C07308=1176.421,-51.106,-43.025,179.479,5.781,149.182
C07309=1176.426,-51.356,-43.013,179.477,5.780,149.183
C07310=1176.431,-51.606,-43.001,179.474,5.780,149.183
C07311=1176.436,-51.856,-42.990,179.472,5.780,149.184
C07312=1176.442,-52.105,-42.979,179.470,5.779,149.185
C07313=1176.447,-52.355,-42.967,179.467,5.779,149.185
C07314=1176.452,-52.605,-42.956,179.465,5.778,149.186
C07315=1176.457,-52.855,-42.944,179.463,5.779,149.187
C07316=1176.462,-53.104,-42.933,179.460,5.778,149.187
C07317=1176.468,-53.354,-42.922,179.458,5.777,149.188
C07318=1176.473,-53.603,-42.910,179.455,5.777,149.188
C07319=1176.477,-53.853,-42.899,179.453,5.777,149.189
C07320=1176.483,-54.103,-42.887,179.451,5.776,149.190
C07321=1176.489,-54.352,-42.877,179.448,5.776,149.190
C07322=1176.494,-54.602,-42.865,179.446,5.776,149.191
C07323=1176.499,-54.852,-42.854,179.444,5.776,149.191
C07324=1176.504,-55.102,-42.842,179.441,5.775,149.192
C07325=1176.509,-55.351,-42.831,179.439,5.774,149.193
C07326=1176.514,-55.600,-42.820,179.437,5.774,149.193
C07327=1176.520,-55.851,-42.808,179.434,5.774,149.194
C07328=1176.524,-56.101,-42.797,179.432,5.774,149.195
C07329=1176.531,-56.350,-42.786,179.430,5.773,149.195
C07330=1176.535,-56.599,-42.774,179.428,5.774,149.196
C07331=1176.540,-56.850,-42.764,179.425,5.773,149.196
C07332=1176.546,-57.099,-42.752,179.423,5.772,149.197
C07333=1176.551,-57.349,-42.741,179.420,5.771,149.198
C07334=1176.556,-57.598,-42.730,179.418,5.772,149.198
C07335=1176.561,-57.849,-42.718,179.416,5.771,149.199
C07336=1176.567,-58.098,-42.708,179.414,5.771,149.199
C07337=1176.572,-58.348,-42.696,179.411,5.770,149.200
C07338=1176.577,-58.597,-42.684,179.409,5.771,149.201
C07339=1176.582,-58.847,-42.674,179.407,5.770,149.201
C07340=1176.588,-59.097,-42.662,179.404,5.769,149.202
C07341=1176.592,-59.346,-42.651,179.402,5.769,149.203
C07342=1176.598,-59.596,-42.641,179.400,5.769,149.203
C07343=1176.603,-59.846,-42.629,179.397,5.769,149.204
C07344=1176.608,-60.095,-42.618,179.395,5.768,149.204
C07345=1176.614,-60.345,-42.607,179.393,5.768,149.205
C07346=1176.618,-60.595,-42.596,179.390,5.768,149.206
C07347=1176.624,-60.845,-42.584,179.388,5.767,149.206
C07348=1176.630,-61.094,-42.574,179.385,5.767,149.207
C07349=1176.634,-61.344,-42.563,179.384,5.766,149.208
C07350=1176.640,-61.594,-42.551,179.381,5.766,149.208
C07351=1176.645,-61.843,-42.541,179.378,5.766,149.209
C07352=1176.650,-62.093,-42.529,179.377,5.766,149.209
C07353=1176.655,-62.343,-42.519,179.374,5.765,149.210
C07354=1176.661,-62.592,-42.507,179.372,5.764,149.211
C07355=1176.666,-62.842,-42.496,179.369,5.764,149.211
C07356=1176.671,-63.092,-42.485,179.367,5.764,149.212
C07357=1176.676,-63.341,-42.474,179.365,5.764,149.212
C07358=1176.682,-63.592,-42.463,179.362,5.763,149.213
C07359=1176.687,-63.841,-42.452,179.360,5.764,149.214
C07360=1176.692,-64.090,-42.441,179.358,5.763,149.214
C07361=1176.697,-64.340,-42.430,179.355,5.762,149.215
C07362=1176.703,-64.590,-42.419,179.354,5.762,149.216
C07363=1176.708,-64.840,-42.408,179.351,5.762,149.216
C07364=1176.712,-65.090,-42.397,179.348,5.762,149.217
C07365=1176.718,-65.339,-42.387,179.346,5.761,149.217
C07366=1176.723,-65.589,-42.376,179.344,5.761,149.218
C07367=1176.729,-65.839,-42.365,179.342,5.760,149.219
C07368=1176.734,-66.088,-42.354,179.339,5.760,149.219
C07369=1176.739,-66.338,-42.343,179.337,5.760,149.220
C07370=1176.744,-66.587,-42.332,179.335,5.759,149.221
C07371=1176.749,-66.838,-42.321,179.332,5.759,149.221
C07372=1176.755,-67.087,-42.310,179.331,5.759,149.222
C07373=1176.760,-67.337,-42.299,179.328,5.759,149.222
C07374=1176.765,-67.586,-42.288,179.325,5.758,149.223
C07375=1176.770,-67.836,-42.278,179.324,5.758,149.224
C07376=1176.776,-68.086,-42.268,179.321,5.758,149.224
C07377=1176.781,-68.335,-42.256,179.319,5.757,149.225
C07378=1176.786,-68.586,-42.245,179.316,5.757,149.225
C07379=1176.792,-68.835,-42.234,179.314,5.757,149.226
C07380=1176.797,-69.085,-42.224,179.312,5.756,149.227
C07381=1176.802,-69.335,-42.213,179.309,5.756,149.227
C07382=1176.807,-69.584,-42.202,179.308,5.756,149.228
C07383=1176.813,-69.834,-42.192,179.305,5.755,149.229
C07384=1176.817,-70.084,-42.181,179.302,5.755,149.229
C07385=1176.823,-70.333,-42.170,179.301,5.755,149.230
C07386=1176.829,-70.584,-42.159,179.298,5.755,149.230
C07387=1176.834,-70.833,-42.148,179.296,5.754,149.231
C07388=1176.839,-71.083,-42.138,179.294,5.754,149.232
C07389=1176.844,-71.332,-42.128,179.291,5.754,149.232
C07390=1176.849,-71.582,-42.116,179.289,5.753,149.233
C07391=1176.855,-71.831,-42.106,179.287,5.753,149.234
C07392=1176.860,-72.082,-42.096,179.285,5.753,149.234
C07393=1176.865,-72.331,-42.085,179.282,5.752,149.235
C07394=1176.870,-72.581,-42.074,179.280,5.753,149.235
C07395=1176.876,-72.830,-42.064,179.278,5.752,149.236
C07396=1176.880,-73.080,-42.053,179.275,5.751,149.237
C07397=1176.886,-73.330,-42.042,179.274,5.751,149.237
C07398=1176.891,-73.580,-42.032,179.271,5.751,149.238
C07399=1176.896,-73.829,-42.021,179.268,5.751,149.239
C07400=1176.902,-74.079,-42.010,179.267,5.751,149.239
C07401=1176.908,-74.329,-41.999,179.264,5.750,149.240
C07402=1176.913,-74.579,-41.989,179.262,5.749,149.240
C07403=1176.918,-74.828,-41.978,179.260,5.750,149.241
C07404=1176.923,-75.078,-41.967,179.257,5.749,149.241
C07405=1176.928,-75.328,-41.957,179.255,5.749,149.242
C07406=1176.934,-75.599,-41.946,179.253,5.749,149.243
C07407=1176.940,-75.869,-41.934,179.250,5.749,149.243
C07408=1176.945,-76.141,-41.923,179.248,5.748,149.244
C07409=1176.951,-76.412,-41.912,179.245,5.747,149.245
C07410=1176.956,-76.661,-41.901,179.243,5.748,149.245
C07411=1176.962,-76.911,-41.891,179.241,5.747,149.246
C07412=1176.967,-77.161,-41.880,179.238,5.747,149.247
C07413=1176.972,-77.411,-41.870,179.236,5.747,149.247
C07414=1176.977,-77.661,-41.859,179.234,5.746,149.248
C07415=1176.983,-77.910,-41.849,179.231,5.746,149.248
C07416=1176.988,-78.160,-41.838,179.230,5.746,149.249
C07417=1176.993,-78.410,-41.828,179.227,5.745,149.250
C07418=1176.999,-78.659,-41.817,179.225,5.745,149.250
C07419=1177.004,-78.909,-41.807,179.223,5.745,149.251
C07420=1177.009,-79.159,-41.797,179.220,5.745,149.252
C07421=1177.014,-79.409,-41.786,179.218,5.744,149.252
C07422=1177.019,-79.658,-41.776,179.216,5.744,149.253
C07423=1177.025,-79.908,-41.766,179.214,5.743,149.253
C07424=1177.030,-80.158,-41.755,179.211,5.743,149.254
C07425=1177.035,-80.407,-41.745,179.209,5.743,149.254
C07426=1177.040,-80.657,-41.734,179.207,5.743,149.255
C07427=1177.046,-80.907,-41.724,179.205,5.743,149.256
C07428=1177.051,-81.156,-41.714,179.202,5.742,149.256
C07429=1177.056,-81.407,-41.703,179.200,5.742,149.257
C07430=1177.062,-81.656,-41.693,179.198,5.742,149.258
C07431=1177.068,-81.906,-41.683,179.196,5.741,149.258
C07432=1177.072,-82.156,-41.673,179.193,5.741,149.259
C07433=1177.077,-82.405,-41.663,179.191,5.741,149.259
C07434=1177.082,-82.655,-41.652,179.189,5.741,149.260
C07435=1177.088,-82.905,-41.642,179.187,5.741,149.261
C07436=1177.094,-83.155,-41.632,179.184,5.740,149.261
C07437=1177.099,-83.405,-41.621,179.182,5.739,149.262
C07438=1177.104,-83.654,-41.611,179.180,5.740,149.263
C07439=1177.109,-83.904,-41.601,179.178,5.739,149.263
C07440=1177.114,-84.154,-41.591,179.175,5.739,149.264
C07441=1177.120,-84.403,-41.580,179.173,5.739,149.264
C07442=1177.125,-84.653,-41.570,179.171,5.738,149.265
C07443=1177.130,-84.903,-41.560,179.169,5.739,149.266
C07444=1177.135,-85.152,-41.550,179.167,5.738,149.266
C07445=1177.141,-85.402,-41.540,179.164,5.737,149.267
C07446=1177.146,-85.652,-41.529,179.162,5.737,149.267
C07447=1177.151,-85.902,-41.519,179.160,5.737,149.268
C07448=1177.157,-86.151,-41.509,179.157,5.736,149.268
C07449=1177.161,-86.401,-41.499,179.155,5.737,149.269
C07450=1177.167,-86.651,-41.489,179.153,5.736,149.270
C07451=1177.172,-86.900,-41.478,179.151,5.736,149.270
C07452=1177.178,-87.150,-41.468,179.148,5.736,149.271
C07453=1177.183,-87.400,-41.459,179.146,5.735,149.272
C07454=1177.188,-87.650,-41.449,179.144,5.735,149.272
C07455=1177.194,-87.899,-41.439,179.142,5.735,149.273
C07456=1177.199,-88.150,-41.428,179.140,5.735,149.273
C07457=1177.204,-88.399,-41.418,179.138,5.734,149.274
C07458=1177.209,-88.648,-41.408,179.135,5.734,149.275
C07459=1177.215,-88.898,-41.398,179.133,5.734,149.275
C07460=1177.220,-89.148,-41.387,179.131,5.733,149.276
C07461=1177.225,-89.398,-41.378,179.129,5.733,149.276
C07462=1177.231,-89.648,-41.368,179.127,5.733,149.277
C07463=1177.236,-89.898,-41.358,179.124,5.733,149.278
C07464=1177.240,-90.147,-41.348,179.122,5.733,149.278
C07465=1177.246,-90.397,-41.338,179.120,5.732,149.279
C07466=1177.252,-90.646,-41.328,179.118,5.732,149.279
C07467=1177.256,-90.897,-41.318,179.115,5.732,149.280
C07468=1177.262,-91.146,-41.308,179.113,5.731,149.281
C07469=1177.267,-91.396,-41.298,179.111,5.732,149.281
C07470=1177.273,-91.645,-41.288,179.109,5.731,149.282
C07471=1177.278,-91.896,-41.278,179.107,5.731,149.283
C07472=1177.283,-92.145,-41.268,179.105,5.730,149.283
C07473=1177.289,-92.395,-41.258,179.102,5.730,149.284
C07474=1177.294,-92.644,-41.248,179.100,5.730,149.284
C07475=1177.300,-92.894,-41.239,179.098,5.730,149.285
C07476=1177.305,-93.145,-41.228,179.096,5.730,149.285
C07477=1177.309,-93.394,-41.219,179.093,5.729,149.286
C07478=1177.315,-93.643,-41.209,179.091,5.729,149.287
C07479=1177.320,-93.893,-41.200,179.089,5.729,149.287
C07480=1177.326,-94.143,-41.189,179.086,5.728,149.288
C07481=1177.331,-94.393,-41.179,179.085,5.728,149.289
C07482=1177.336,-94.642,-41.169,179.082,5.728,149.289
C07483=1177.342,-94.892,-41.160,179.081,5.728,149.290
C07484=1177.347,-95.142,-41.150,179.078,5.728,149.290
C07485=1177.352,-95.391,-41.140,179.076,5.727,149.291
C07486=1177.357,-95.642,-41.130,179.074,5.727,149.292
C07487=1177.362,-95.891,-41.120,179.071,5.726,149.292
C07488=1177.368,-96.141,-41.110,179.069,5.727,149.293
C07489=1177.374,-96.391,-41.101,179.067,5.726,149.293
C07490=1177.379,-96.640,-41.091,179.064,5.726,149.294
C07491=1177.384,-96.890,-41.081,179.063,5.726,149.294
C07492=1177.389,-97.140,-41.072,179.060,5.725,149.295
C07493=1177.394,-97.390,-41.061,179.059,5.725,149.296
C07494=1177.399,-97.640,-41.053,179.056,5.725,149.296
C07495=1177.405,-97.889,-41.042,179.054,5.725,149.297
C07496=1177.411,-98.139,-41.032,179.052,5.725,149.298
C07497=1177.416,-98.389,-41.023,179.049,5.724,149.298
C07498=1177.421,-98.639,-41.013,179.047,5.724,149.299
C07499=1177.426,-98.889,-41.004,179.045,5.723,149.299
C07500=1177.432,-99.138,-40.994,179.043,5.724,149.300
C07501=1177.436,-99.388,-40.984,179.041,5.723,149.300
C07502=1177.442,-99.638,-40.974,179.039,5.723,149.301
C07503=1177.447,-99.887,-40.965,179.037,5.723,149.302
C07504=1177.453,-100.137,-40.955,179.034,5.722,149.302
C07505=1177.458,-100.386,-40.946,179.032,5.722,149.303
C07506=1177.463,-100.637,-40.936,179.030,5.722,149.304
C07507=1177.468,-100.886,-40.926,179.028,5.722,149.304
C07508=1177.474,-101.137,-40.917,179.025,5.722,149.305
C07509=1177.479,-101.386,-40.907,179.024,5.722,149.305
C07510=1177.485,-101.658,-40.896,179.021,5.721,149.306
C07511=1177.491,-101.930,-40.886,179.018,5.721,149.307
C07512=1177.497,-102.201,-40.876,179.016,5.721,149.307
C07513=1177.502,-102.473,-40.865,179.014,5.720,149.308
C07514=1177.508,-102.723,-40.856,179.012,5.720,149.309
C07515=1177.513,-102.972,-40.846,179.010,5.720,149.309
C07516=1177.519,-103.222,-40.837,179.007,5.720,149.310
C07517=1177.523,-103.471,-40.827,179.006,5.720,149.310
C07518=1177.529,-103.722,-40.817,179.003,5.719,149.311
C07519=1177.534,-103.972,-40.808,179.001,5.719,149.311
C07520=1177.539,-104.221,-40.799,178.999,5.719,149.312
C07521=1177.545,-104.471,-40.789,178.996,5.718,149.313
C07522=1177.550,-104.721,-40.780,178.994,5.719,149.313
C07523=1177.555,-104.971,-40.770,178.992,5.718,149.314
C07524=1177.560,-105.220,-40.761,178.990,5.718,149.315
C07525=1177.566,-105.470,-40.751,178.988,5.717,149.315
C07526=1177.571,-105.720,-40.742,178.986,5.718,149.316
C07527=1177.576,-105.969,-40.733,178.984,5.717,149.316
C07528=1177.582,-106.219,-40.723,178.982,5.717,149.317
C07529=1177.587,-106.469,-40.713,178.979,5.717,149.317
C07530=1177.593,-106.719,-40.704,178.978,5.717,149.318
C07531=1177.598,-106.969,-40.695,178.975,5.716,149.319
C07532=1177.603,-107.218,-40.685,178.973,5.716,149.319
C07533=1177.609,-107.468,-40.676,178.971,5.716,149.320
C07534=1177.614,-107.718,-40.667,178.969,5.715,149.320
C07535=1177.619,-107.967,-40.657,178.967,5.716,149.321
C07536=1177.625,-108.217,-40.648,178.964,5.715,149.322
C07537=1177.630,-108.467,-40.639,178.962,5.715,149.322
C07538=1177.635,-108.716,-40.629,178.960,5.714,149.323
C07539=1177.641,-108.967,-40.620,178.958,5.715,149.323
C07540=1177.646,-109.216,-40.611,178.956,5.714,149.324
C07541=1177.651,-109.466,-40.601,178.954,5.714,149.325
C07542=1177.657,-109.716,-40.592,178.952,5.714,149.325
C07543=1177.662,-109.966,-40.583,178.950,5.714,149.326
C07544=1177.667,-110.215,-40.573,178.947,5.713,149.326
C07545=1177.673,-110.465,-40.564,178.946,5.713,149.327
C07546=1177.678,-110.715,-40.555,178.943,5.713,149.328
C07547=1177.683,-110.965,-40.546,178.941,5.712,149.328
C07548=1177.688,-111.214,-40.536,178.939,5.713,149.329
C07549=1177.694,-111.464,-40.527,178.937,5.712,149.329
C07550=1177.699,-111.714,-40.518,178.934,5.712,149.330
C07551=1177.705,-111.964,-40.509,178.932,5.711,149.330
C07552=1177.710,-112.213,-40.499,178.930,5.712,149.331
C07553=1177.715,-112.463,-40.490,178.928,5.711,149.332
C07554=1177.720,-112.713,-40.481,178.926,5.711,149.332
C07555=1177.726,-112.963,-40.472,178.924,5.711,149.333
C07556=1177.731,-113.213,-40.462,178.922,5.711,149.333
C07557=1177.736,-113.462,-40.453,178.919,5.710,149.334
C07558=1177.742,-113.713,-40.444,178.918,5.710,149.335
C07559=1177.747,-113.962,-40.435,178.915,5.710,149.335
C07560=1177.752,-114.212,-40.426,178.914,5.710,149.336
C07561=1177.757,-114.462,-40.417,178.911,5.710,149.336
C07562=1177.763,-114.712,-40.407,178.909,5.710,149.337
C07563=1177.768,-114.961,-40.398,178.907,5.709,149.337
C07564=1177.773,-115.211,-40.389,178.905,5.709,149.338
C07565=1177.778,-115.461,-40.380,178.903,5.709,149.339
C07566=1177.784,-115.710,-40.372,178.901,5.709,149.339
C07567=1177.790,-115.961,-40.362,178.899,5.708,149.340
C07568=1177.795,-116.210,-40.352,178.896,5.709,149.341
C07569=1177.800,-116.460,-40.344,178.894,5.708,149.341
C07570=1177.805,-116.709,-40.335,178.893,5.708,149.342
C07571=1177.810,-116.959,-40.326,178.890,5.707,149.342
C07572=1177.816,-117.209,-40.316,178.888,5.708,149.343
C07573=1177.821,-117.459,-40.307,178.886,5.707,149.343
C07574=1177.827,-117.709,-40.298,178.884,5.707,149.344
C07575=1177.832,-117.959,-40.290,178.881,5.707,149.345
C07576=1177.837,-118.209,-40.281,178.879,5.706,149.345
C07577=1177.843,-118.458,-40.272,178.878,5.706,149.346
C07578=1177.849,-118.708,-40.263,178.875,5.706,149.346
C07579=1177.853,-118.957,-40.253,178.873,5.706,149.347
C07580=1177.859,-119.207,-40.244,178.871,5.705,149.348
C07581=1177.864,-119.457,-40.235,178.869,5.705,149.348
C07582=1177.869,-119.707,-40.226,178.866,5.705,149.349
C07583=1177.874,-119.957,-40.217,178.865,5.705,149.349
C07584=1177.880,-120.207,-40.208,178.863,5.704,149.350
C07585=1177.886,-120.456,-40.199,178.861,5.705,149.350
C07586=1177.891,-120.706,-40.191,178.858,5.704,149.351
C07587=1177.896,-120.956,-40.182,178.856,5.704,149.352
C07588=1177.901,-121.206,-40.173,178.854,5.703,149.352
C07589=1177.906,-121.456,-40.164,178.852,5.704,149.353
C07590=1177.912,-121.705,-40.155,178.850,5.704,149.353
C07591=1177.917,-121.955,-40.146,178.848,5.703,149.354
C07592=1177.923,-122.204,-40.138,178.846,5.704,149.354
C07593=1177.928,-122.455,-40.128,178.844,5.703,149.355
C07594=1177.934,-122.704,-40.119,178.842,5.703,149.355
C07595=1177.939,-122.954,-40.110,178.840,5.702,149.356
C07596=1177.944,-123.204,-40.101,178.838,5.702,149.357
C07597=1177.949,-123.454,-40.092,178.835,5.702,149.357
C07598=1177.955,-123.704,-40.085,178.834,5.702,149.358
C07599=1177.960,-123.954,-40.076,178.832,5.701,149.358
C07600=1177.966,-124.203,-40.067,178.829,5.702,149.359
C07601=1177.971,-124.453,-40.058,178.827,5.701,149.360
C07602=1177.976,-124.703,-40.049,178.825,5.701,149.360
C07603=1177.981,-124.953,-40.040,178.823,5.701,149.361
C07604=1177.987,-125.202,-40.032,178.821,5.701,149.361
C07605=1177.992,-125.452,-40.023,178.819,5.700,149.362
C07606=1177.997,-125.702,-40.014,178.817,5.700,149.362
C07607=1178.002,-125.952,-40.005,178.815,5.700,149.363
C07608=1178.008,-126.201,-39.996,178.813,5.700,149.364
C07609=1178.014,-126.451,-39.988,178.811,5.699,149.364
C07610=1178.019,-126.701,-39.979,178.809,5.700,149.365
C07611=1178.024,-126.951,-39.970,178.806,5.699,149.365
C07612=1178.029,-127.201,-39.961,178.805,5.699,149.366
C07613=1178.035,-127.450,-39.953,178.802,5.699,149.367
C07614=1177.614,-127.462,-39.992,178.799,5.703,149.368
C07615=1177.609,-127.212,-40.001,178.801,5.702,149.368
C07616=1177.604,-126.962,-40.010,178.803,5.703,149.367
C07617=1177.598,-126.712,-40.019,178.805,5.703,149.367
C07618=1177.593,-126.463,-40.028,178.807,5.702,149.366
C07619=1177.587,-126.213,-40.037,178.809,5.703,149.366
C07620=1177.581,-125.962,-40.045,178.811,5.703,149.365
C07621=1177.576,-125.712,-40.054,178.813,5.704,149.364
C07622=1177.570,-125.463,-40.063,178.815,5.704,149.364
C07623=1177.565,-125.213,-40.072,178.818,5.704,149.363
C07624=1177.560,-124.964,-40.081,178.819,5.704,149.363
C07625=1177.555,-124.714,-40.089,178.821,5.705,149.362
C07626=1177.550,-124.464,-40.098,178.823,5.704,149.361
C07627=1177.544,-124.215,-40.107,178.826,5.705,149.361
C07628=1177.539,-123.965,-40.116,178.828,5.705,149.360
C07629=1177.533,-123.715,-40.125,178.830,5.705,149.360
C07630=1177.528,-123.465,-40.134,178.831,5.705,149.359
C07631=1177.523,-123.215,-40.142,178.834,5.706,149.359
C07632=1177.518,-122.965,-40.151,178.836,5.706,149.358
C07633=1177.512,-122.716,-40.159,178.838,5.706,149.357
C07634=1177.507,-122.466,-40.168,178.840,5.706,149.357
C07635=1177.502,-122.216,-40.177,178.842,5.707,149.356
C07636=1177.496,-121.966,-40.186,178.844,5.706,149.356
C07637=1177.491,-121.716,-40.195,178.846,5.707,149.355
C07638=1177.485,-121.466,-40.204,178.848,5.707,149.355
C07639=1177.480,-121.217,-40.213,178.851,5.708,149.354
C07640=1177.474,-120.967,-40.222,178.852,5.707,149.353
C07641=1177.469,-120.717,-40.231,178.855,5.708,149.353
C07642=1177.464,-120.467,-40.240,178.857,5.708,149.352
C07643=1177.459,-120.218,-40.248,178.859,5.708,149.352
C07644=1177.454,-119.968,-40.257,178.861,5.708,149.351
C07645=1177.448,-119.718,-40.267,178.863,5.709,149.351
C07646=1177.443,-119.468,-40.276,178.865,5.709,149.350
C07647=1177.437,-119.219,-40.284,178.867,5.709,149.349
C07648=1177.432,-118.969,-40.293,178.869,5.709,149.349
C07649=1177.427,-118.719,-40.303,178.872,5.710,149.348
C07650=1177.422,-118.470,-40.312,178.873,5.710,149.348
C07651=1177.417,-118.220,-40.321,178.876,5.710,149.347
C07652=1177.411,-117.970,-40.330,178.878,5.710,149.346
C07653=1177.405,-117.720,-40.339,178.880,5.710,149.346
C07654=1177.400,-117.470,-40.348,178.882,5.710,149.345
C07655=1177.395,-117.220,-40.357,178.884,5.711,149.345
C07656=1177.389,-116.971,-40.365,178.886,5.711,149.344
C07657=1177.384,-116.721,-40.374,178.888,5.711,149.344
C07658=1177.378,-116.471,-40.384,178.890,5.711,149.343
C07659=1177.373,-116.221,-40.393,178.893,5.712,149.342
C07660=1177.368,-115.972,-40.402,178.895,5.711,149.342
C07661=1177.363,-115.722,-40.411,178.897,5.712,149.341
C07662=1177.357,-115.472,-40.421,178.898,5.712,149.341
C07663=1177.352,-115.222,-40.429,178.901,5.713,149.340
C07664=1177.347,-114.972,-40.438,178.903,5.713,149.339
C07665=1177.342,-114.722,-40.447,178.905,5.713,149.339
C07666=1177.337,-114.472,-40.456,178.907,5.713,149.338
C07667=1177.331,-114.223,-40.466,178.910,5.713,149.338
C07668=1177.325,-113.974,-40.475,178.911,5.713,149.337
C07669=1177.320,-113.724,-40.484,178.914,5.714,149.336
C07670=1177.315,-113.474,-40.493,178.916,5.714,149.336
C07671=1177.309,-113.224,-40.502,178.918,5.714,149.335
C07672=1177.304,-112.975,-40.512,178.920,5.714,149.335
C07673=1177.299,-112.725,-40.521,178.922,5.715,149.334
C07674=1177.293,-112.475,-40.530,178.925,5.715,149.333
C07675=1177.288,-112.225,-40.539,178.926,5.715,149.333
C07676=1177.283,-111.975,-40.548,178.929,5.715,149.332
C07677=1177.278,-111.726,-40.558,178.931,5.715,149.332
C07678=1177.272,-111.475,-40.567,178.933,5.716,149.331
C07679=1177.267,-111.226,-40.576,178.935,5.716,149.331
C07680=1177.262,-110.976,-40.585,178.937,5.717,149.330
C07681=1177.256,-110.726,-40.595,178.939,5.716,149.329
C07682=1177.251,-110.476,-40.604,178.941,5.717,149.329
C07683=1177.246,-110.227,-40.613,178.943,5.717,149.328
C07684=1177.240,-109.976,-40.622,178.946,5.717,149.328
C07685=1177.235,-109.727,-40.632,178.948,5.717,149.327
C07686=1177.230,-109.477,-40.641,178.950,5.718,149.327
C07687=1177.224,-109.227,-40.650,178.952,5.717,149.326
C07688=1177.219,-108.978,-40.660,178.954,5.718,149.325
C07689=1177.214,-108.728,-40.669,178.956,5.718,149.325
C07690=1177.208,-108.478,-40.678,178.958,5.718,149.324
C07691=1177.203,-108.229,-40.688,178.961,5.719,149.324
C07692=1177.198,-107.979,-40.697,178.963,5.719,149.323
C07693=1177.192,-107.729,-40.706,178.965,5.720,149.322
C07694=1177.187,-107.479,-40.716,178.967,5.719,149.322
C07695=1177.182,-107.230,-40.725,178.969,5.720,149.321
C07696=1177.176,-106.979,-40.734,178.971,5.719,149.321
C07697=1177.171,-106.730,-40.744,178.973,5.720,149.320
C07698=1177.166,-106.480,-40.753,178.976,5.720,149.319
C07699=1177.160,-106.231,-40.763,178.978,5.721,149.319
C07700=1177.155,-105.981,-40.772,178.980,5.720,149.318
C07701=1177.149,-105.731,-40.781,178.982,5.721,149.318
C07702=1177.144,-105.482,-40.791,178.985,5.721,149.317
C07703=1177.139,-105.232,-40.800,178.986,5.721,149.316
C07704=1177.134,-104.982,-40.810,178.989,5.722,149.316
C07705=1177.129,-104.732,-40.819,178.991,5.722,149.315
C07706=1177.123,-104.481,-40.829,178.993,5.723,149.315
C07707=1177.118,-104.232,-40.839,178.995,5.722,149.314
C07708=1177.112,-103.982,-40.848,178.997,5.723,149.314
C07709=1177.108,-103.733,-40.858,178.999,5.722,149.313
C07710=1177.102,-103.483,-40.867,179.001,5.723,149.312
C07711=1177.097,-103.233,-40.877,179.003,5.723,149.312
C07712=1177.092,-102.984,-40.886,179.006,5.724,149.311
C07713=1177.086,-102.734,-40.896,179.008,5.724,149.310
C07714=1177.081,-102.484,-40.905,179.010,5.724,149.310
C07715=1177.075,-102.212,-40.915,179.012,5.724,149.309
C07716=1177.069,-101.940,-40.926,179.015,5.725,149.309
C07717=1177.064,-101.669,-40.937,179.017,5.725,149.308
C07718=1177.058,-101.397,-40.947,179.019,5.725,149.307
C07719=1177.052,-101.147,-40.956,179.022,5.725,149.307
C07720=1177.048,-100.897,-40.966,179.024,5.726,149.306
C07721=1177.042,-100.647,-40.976,179.026,5.726,149.305
C07722=1177.037,-100.398,-40.985,179.028,5.726,149.305
C07723=1177.031,-100.148,-40.995,179.031,5.726,149.304
C07724=1177.026,-99.899,-41.004,179.032,5.726,149.304
C07725=1177.020,-99.648,-41.014,179.035,5.727,149.303
C07726=1177.015,-99.399,-41.023,179.037,5.727,149.303
C07727=1177.010,-99.150,-41.034,179.039,5.727,149.302
C07728=1177.005,-98.899,-41.043,179.041,5.728,149.301
C07729=1177.000,-98.650,-41.053,179.043,5.727,149.301
C07730=1176.995,-98.400,-41.062,179.046,5.728,149.300
C07731=1176.989,-98.150,-41.072,179.048,5.728,149.299
C07732=1176.984,-97.900,-41.081,179.050,5.729,149.299
C07733=1176.978,-97.651,-41.091,179.052,5.728,149.298
C07734=1176.973,-97.401,-41.102,179.054,5.729,149.298
C07735=1176.968,-97.151,-41.111,179.057,5.729,149.297
C07736=1176.962,-96.901,-41.121,179.058,5.729,149.297
C07737=1176.958,-96.652,-41.131,179.061,5.730,149.296
C07738=1176.952,-96.402,-41.140,179.063,5.730,149.295
C07739=1176.947,-96.152,-41.150,179.065,5.730,149.295
C07740=1176.941,-95.903,-41.160,179.067,5.730,149.294
C07741=1176.936,-95.652,-41.170,179.070,5.730,149.293
C07742=1176.931,-95.403,-41.179,179.072,5.731,149.293
C07743=1176.925,-95.153,-41.190,179.074,5.731,149.292
C07744=1176.920,-94.903,-41.199,179.076,5.732,149.292
C07745=1176.915,-94.654,-41.209,179.078,5.731,149.291
C07746=1176.910,-94.404,-41.219,179.080,5.732,149.291
C07747=1176.904,-94.154,-41.228,179.083,5.732,149.290
C07748=1176.899,-93.904,-41.238,179.085,5.732,149.289
C07749=1176.893,-93.655,-41.249,179.087,5.733,149.289
C07750=1176.888,-93.405,-41.258,179.089,5.733,149.288
C07751=1176.883,-93.155,-41.268,179.092,5.733,149.287
C07752=1176.878,-92.905,-41.278,179.093,5.733,149.287
C07753=1176.873,-92.656,-41.288,179.096,5.734,149.286
C07754=1176.867,-92.406,-41.297,179.098,5.734,149.286
C07755=1176.861,-92.156,-41.308,179.100,5.734,149.285
C07756=1176.857,-91.906,-41.318,179.103,5.734,149.284
C07757=1176.851,-91.657,-41.328,179.104,5.734,149.284
C07758=1176.845,-91.406,-41.337,179.107,5.735,149.283
C07759=1176.841,-91.157,-41.347,179.109,5.735,149.283
C07760=1176.836,-90.907,-41.357,179.111,5.735,149.282
C07761=1176.830,-90.657,-41.368,179.114,5.736,149.282
C07762=1176.825,-90.408,-41.377,179.116,5.735,149.281
C07763=1176.819,-90.158,-41.387,179.118,5.736,149.280
C07764=1176.814,-89.908,-41.397,179.121,5.737,149.280
C07765=1176.809,-89.659,-41.407,179.122,5.737,149.279
C07766=1176.804,-89.409,-41.417,179.125,5.737,149.278
C07767=1176.798,-89.160,-41.427,179.126,5.737,149.278
C07768=1176.793,-88.909,-41.438,179.129,5.737,149.277
C07769=1176.788,-88.659,-41.447,179.131,5.738,149.277
C07770=1176.782,-88.410,-41.457,179.133,5.738,149.276
C07771=1176.777,-88.160,-41.468,179.136,5.738,149.275
C07772=1176.773,-87.910,-41.477,179.138,5.738,149.275
C07773=1176.767,-87.661,-41.487,179.140,5.739,149.274
C07774=1176.761,-87.411,-41.498,179.143,5.739,149.274
C07775=1176.756,-87.161,-41.508,179.145,5.739,149.273
C07776=1176.751,-86.912,-41.518,179.147,5.740,149.272
C07777=1176.746,-86.662,-41.528,179.149,5.740,149.272
C07778=1176.741,-86.411,-41.538,179.151,5.740,149.271
C07779=1176.735,-86.162,-41.548,179.154,5.741,149.271
C07780=1176.729,-85.912,-41.558,179.155,5.741,149.270
C07781=1176.725,-85.662,-41.568,179.158,5.741,149.269
C07782=1176.719,-85.413,-41.579,179.161,5.741,149.269
C07783=1176.714,-85.163,-41.589,179.162,5.741,149.268
C07784=1176.708,-84.914,-41.599,179.165,5.742,149.267
C07785=1176.703,-84.664,-41.610,179.167,5.742,149.267
C07786=1176.698,-84.414,-41.619,179.169,5.742,149.266
C07787=1176.693,-84.165,-41.629,179.171,5.743,149.266
C07788=1176.688,-83.915,-41.640,179.173,5.743,149.265
C07789=1176.682,-83.665,-41.650,179.176,5.743,149.265
C07790=1176.677,-83.415,-41.661,179.178,5.744,149.264
C07791=1176.672,-83.165,-41.670,179.180,5.743,149.263
C07792=1176.667,-82.916,-41.681,179.183,5.744,149.263
C07793=1176.662,-82.666,-41.691,179.185,5.744,149.262
C07794=1176.656,-82.416,-41.701,179.187,5.744,149.262
C07795=1176.651,-82.167,-41.712,179.190,5.745,149.261
C07796=1176.646,-81.916,-41.722,179.191,5.745,149.260
C07797=1176.640,-81.667,-41.732,179.194,5.745,149.260
C07798=1176.635,-81.418,-41.742,179.196,5.746,149.259
C07799=1176.630,-81.167,-41.753,179.198,5.746,149.258
C07800=1176.625,-80.918,-41.763,179.201,5.746,149.258
C07801=1176.620,-80.668,-41.773,179.203,5.747,149.257
C07802=1176.614,-80.418,-41.784,179.205,5.746,149.257
C07803=1176.609,-80.169,-41.794,179.207,5.747,149.256
C07804=1176.604,-79.919,-41.805,179.209,5.747,149.255
C07805=1176.598,-79.669,-41.815,179.211,5.748,149.255
C07806=1176.592,-79.420,-41.825,179.214,5.748,149.254
C07807=1176.587,-79.170,-41.836,179.216,5.748,149.253
C07808=1176.583,-78.920,-41.846,179.218,5.748,149.253
C07809=1176.578,-78.670,-41.856,179.221,5.749,149.252
C07810=1176.572,-78.421,-41.866,179.223,5.749,149.252
C07811=1176.566,-78.171,-41.877,179.225,5.749,149.251
C07812=1176.562,-77.921,-41.888,179.228,5.750,149.251
C07813=1176.556,-77.672,-41.898,179.230,5.750,149.250
C07814=1176.551,-77.422,-41.909,179.232,5.750,149.249
C07815=1176.546,-77.172,-41.919,179.234,5.751,149.249
C07816=1176.541,-76.922,-41.929,179.237,5.750,149.248
C07817=1176.535,-76.672,-41.940,179.239,5.751,149.247
C07818=1176.530,-76.423,-41.951,179.241,5.752,149.247
C07819=1176.524,-76.152,-41.962,179.243,5.751,149.246
C07820=1176.519,-75.880,-41.973,179.246,5.752,149.246
C07821=1176.512,-75.610,-41.985,179.248,5.752,149.245
C07822=1176.507,-75.339,-41.996,179.251,5.753,149.244
C07823=1176.501,-75.088,-42.007,179.253,5.752,149.243
C07824=1176.496,-74.839,-42.017,179.255,5.753,149.243
C07825=1176.490,-74.590,-42.028,179.258,5.754,149.242
C07826=1176.485,-74.340,-42.039,179.260,5.754,149.242
C07827=1176.480,-74.090,-42.049,179.262,5.754,149.241
C07828=1176.475,-73.840,-42.060,179.265,5.754,149.240
C07829=1176.470,-73.591,-42.070,179.266,5.754,149.240
C07830=1176.465,-73.341,-42.081,179.269,5.755,149.239
C07831=1176.459,-73.091,-42.091,179.271,5.756,149.239
C07832=1176.454,-72.841,-42.103,179.273,5.755,149.238
C07833=1176.449,-72.592,-42.113,179.276,5.756,149.238
C07834=1176.444,-72.342,-42.123,179.278,5.756,149.237
C07835=1176.438,-72.092,-42.134,179.280,5.756,149.236
C07836=1176.433,-71.842,-42.145,179.283,5.757,149.236
C07837=1176.428,-71.593,-42.155,179.285,5.757,149.235
C07838=1176.423,-71.343,-42.166,179.287,5.757,149.234
C07839=1176.418,-71.094,-42.177,179.289,5.758,149.234
C07840=1176.413,-70.844,-42.187,179.292,5.758,149.233
C07841=1176.406,-70.594,-42.198,179.294,5.758,149.233
C07842=1176.402,-70.344,-42.209,179.296,5.759,149.232
C07843=1176.396,-70.094,-42.219,179.299,5.759,149.231
C07844=1176.391,-69.845,-42.231,179.301,5.759,149.231
C07845=1176.386,-69.595,-42.241,179.303,5.759,149.230
C07846=1176.381,-69.345,-42.251,179.306,5.760,149.229
C07847=1176.375,-69.096,-42.262,179.308,5.760,149.229
C07848=1176.370,-68.846,-42.273,179.310,5.761,149.228
C07849=1176.364,-68.597,-42.285,179.312,5.761,149.228
C07850=1176.359,-68.346,-42.295,179.315,5.761,149.227
C07851=1176.354,-68.096,-42.306,179.317,5.761,149.226
C07852=1176.349,-67.847,-42.317,179.319,5.762,149.226
C07853=1176.344,-67.597,-42.327,179.322,5.763,149.225
C07854=1176.339,-67.348,-42.338,179.324,5.762,149.224
C07855=1176.334,-67.098,-42.349,179.326,5.763,149.224
C07856=1176.328,-66.849,-42.360,179.329,5.763,149.223
C07857=1176.323,-66.598,-42.371,179.331,5.763,149.223
C07858=1176.317,-66.349,-42.382,179.333,5.764,149.222
C07859=1176.312,-66.099,-42.392,179.335,5.764,149.221
C07860=1176.308,-65.850,-42.404,179.338,5.764,149.221
C07861=1176.301,-65.600,-42.414,179.340,5.765,149.220
C07862=1176.297,-65.350,-42.426,179.342,5.765,149.220
C07863=1176.291,-65.101,-42.436,179.345,5.766,149.219
C07864=1176.286,-64.851,-42.447,179.347,5.765,149.218
C07865=1176.281,-64.601,-42.458,179.349,5.766,149.218
C07866=1176.275,-64.351,-42.469,179.352,5.767,149.217
C07867=1176.270,-64.101,-42.480,179.354,5.766,149.216
C07868=1176.265,-63.852,-42.491,179.356,5.767,149.216
C07869=1176.260,-63.602,-42.501,179.358,5.768,149.215
C07870=1176.255,-63.352,-42.513,179.361,5.767,149.215
C07871=1176.249,-63.103,-42.523,179.363,5.768,149.214
C07872=1176.244,-62.853,-42.535,179.365,5.768,149.213
C07873=1176.240,-62.603,-42.546,179.368,5.769,149.213
C07874=1176.233,-62.353,-42.557,179.370,5.769,149.212
C07875=1176.229,-62.104,-42.568,179.372,5.769,149.211
C07876=1176.223,-61.854,-42.578,179.375,5.770,149.211
C07877=1176.218,-61.605,-42.590,179.377,5.770,149.210
C07878=1176.213,-61.355,-42.601,179.379,5.770,149.210
C07879=1176.207,-61.105,-42.612,179.381,5.771,149.209
C07880=1176.203,-60.856,-42.623,179.384,5.771,149.208
C07881=1176.197,-60.606,-42.635,179.386,5.771,149.208
C07882=1176.192,-60.356,-42.645,179.388,5.772,149.207
C07883=1176.187,-60.106,-42.656,179.391,5.772,149.207
C07884=1176.182,-59.857,-42.668,179.393,5.772,149.206
C07885=1176.176,-59.607,-42.678,179.395,5.773,149.205
C07886=1176.171,-59.357,-42.690,179.397,5.773,149.205
C07887=1176.167,-59.108,-42.701,179.400,5.774,149.204
C07888=1176.160,-58.858,-42.712,179.402,5.773,149.203
C07889=1176.155,-58.608,-42.723,179.404,5.774,149.203
C07890=1176.151,-58.359,-42.734,179.407,5.775,149.202
C07891=1176.145,-58.108,-42.746,179.410,5.775,149.202
C07892=1176.140,-57.859,-42.756,179.411,5.775,149.201
C07893=1176.135,-57.609,-42.768,179.414,5.775,149.200
C07894=1176.130,-57.360,-42.780,179.416,5.776,149.200
C07895=1176.124,-57.110,-42.790,179.418,5.776,149.199
C07896=1176.119,-56.860,-42.802,179.421,5.776,149.198
C07897=1176.114,-56.610,-42.813,179.423,5.777,149.198
C07898=1176.109,-56.361,-42.824,179.426,5.777,149.197
C07899=1176.103,-56.111,-42.835,179.428,5.777,149.197
C07900=1176.098,-55.861,-42.846,179.430,5.778,149.196
C07901=1176.094,-55.612,-42.858,179.433,5.778,149.195
C07902=1176.087,-55.362,-42.869,179.435,5.779,149.195
C07903=1176.083,-55.113,-42.881,179.437,5.779,149.194
C07904=1176.077,-54.862,-42.892,179.440,5.779,149.194
C07905=1176.072,-54.613,-42.903,179.442,5.780,149.193
C07906=1176.066,-54.363,-42.915,179.445,5.780,149.192
C07907=1176.062,-54.114,-42.926,179.447,5.780,149.192
C07908=1176.057,-53.864,-42.937,179.449,5.781,149.191
C07909=1176.052,-53.614,-42.949,179.451,5.781,149.190
C07910=1176.046,-53.365,-42.959,179.454,5.782,149.190
C07911=1176.040,-53.115,-42.971,179.456,5.782,149.189
C07912=1176.036,-52.865,-42.982,179.458,5.782,149.189
C07913=1176.030,-52.615,-42.994,179.461,5.783,149.188
C07914=1176.026,-52.366,-43.006,179.463,5.783,149.187
C07915=1176.020,-52.116,-43.017,179.465,5.783,149.187
C07916=1176.015,-51.867,-43.028,179.467,5.784,149.186
C07917=1176.010,-51.617,-43.040,179.470,5.784,149.186
C07918=1176.005,-51.367,-43.052,179.472,5.785,149.185
C07919=1175.999,-51.118,-43.063,179.474,5.785,149.184
C07920=1175.994,-50.868,-43.074,179.477,5.785,149.184
C07921=1175.988,-50.618,-43.085,179.479,5.786,149.183
C07922=1175.984,-50.368,-43.097,179.482,5.786,149.182
C07923=1175.978,-50.098,-43.109,179.485,5.787,149.182
C07924=1175.972,-49.827,-43.122,179.487,5.787,149.181
C07925=1175.967,-49.557,-43.135,179.489,5.787,149.180
C07926=1175.961,-49.287,-43.146,179.491,5.788,149.180
C07927=1175.956,-49.037,-43.158,179.494,5.788,149.179
C07928=1175.951,-48.787,-43.170,179.497,5.788,149.178
C07929=1175.945,-48.537,-43.182,179.499,5.789,149.178
C07930=1175.940,-48.288,-43.193,179.501,5.789,149.177
C07931=1175.934,-48.039,-43.204,179.504,5.789,149.177
C07932=1175.930,-47.789,-43.216,179.506,5.790,149.176
C07933=1175.924,-47.539,-43.228,179.509,5.790,149.175
C07934=1175.920,-47.290,-43.240,179.511,5.791,149.175
C07935=1175.914,-47.040,-43.251,179.513,5.791,149.174
C07936=1175.909,-46.790,-43.263,179.516,5.791,149.174
C07937=1175.904,-46.540,-43.275,179.518,5.792,149.173
C07938=1175.898,-46.291,-43.286,179.520,5.793,149.172
C07939=1175.894,-46.042,-43.297,179.522,5.792,149.172
C07940=1175.888,-45.792,-43.309,179.525,5.793,149.171
C07941=1175.883,-45.542,-43.321,179.527,5.793,149.170
C07942=1175.878,-45.292,-43.332,179.530,5.794,149.170
C07943=1175.873,-45.042,-43.344,179.532,5.795,149.169
C07944=1175.867,-44.792,-43.356,179.534,5.794,149.169
C07945=1175.862,-44.543,-43.368,179.537,5.795,149.168
C07946=1175.857,-44.294,-43.380,179.539,5.796,149.167
C07947=1175.852,-44.044,-43.391,179.542,5.796,149.167
C07948=1175.847,-43.794,-43.403,179.544,5.796,149.166
C07949=1175.841,-43.544,-43.415,179.546,5.796,149.166
C07950=1175.837,-43.295,-43.426,179.549,5.797,149.165
C07951=1175.831,-43.045,-43.438,179.551,5.798,149.164
C07952=1175.826,-42.795,-43.450,179.554,5.798,149.164
C07953=1175.821,-42.546,-43.462,179.556,5.799,149.163
C07954=1175.816,-42.296,-43.474,179.558,5.799,149.162
C07955=1175.810,-42.046,-43.486,179.560,5.799,149.162
C07956=1175.805,-41.796,-43.498,179.563,5.799,149.161
C07957=1175.800,-41.547,-43.508,179.565,5.800,149.161
C07958=1175.795,-41.298,-43.521,179.568,5.801,149.160
C07959=1175.789,-41.048,-43.533,179.570,5.800,149.159
C07960=1175.784,-40.798,-43.544,179.572,5.801,149.159
C07961=1175.779,-40.548,-43.556,179.575,5.802,149.158
C07962=1175.774,-40.299,-43.569,179.578,5.802,149.157
C07963=1175.768,-40.049,-43.581,179.580,5.803,149.157
C07964=1175.764,-39.800,-43.592,179.582,5.802,149.156
C07965=1175.758,-39.550,-43.604,179.584,5.803,149.156
C07966=1175.753,-39.300,-43.616,179.587,5.804,149.155
C07967=1175.748,-39.050,-43.628,179.589,5.804,149.154
C07968=1175.743,-38.801,-43.640,179.591,5.805,149.154
C07969=1175.738,-38.551,-43.652,179.594,5.805,149.153
C07970=1175.733,-38.301,-43.664,179.596,5.805,149.152
C07971=1175.727,-38.052,-43.676,179.598,5.806,149.152
C07972=1175.722,-37.802,-43.688,179.601,5.806,149.151
C07973=1175.717,-37.553,-43.700,179.604,5.807,149.151
C07974=1175.712,-37.303,-43.712,179.606,5.807,149.150
C07975=1175.706,-37.053,-43.724,179.608,5.807,149.149
C07976=1175.701,-36.803,-43.736,179.611,5.808,149.149
C07977=1175.696,-36.553,-43.748,179.613,5.808,149.148
C07978=1175.691,-36.304,-43.760,179.615,5.809,149.147
C07979=1175.686,-36.055,-43.772,179.618,5.809,149.147
C07980=1175.681,-35.805,-43.784,179.620,5.810,149.146
C07981=1175.676,-35.555,-43.796,179.622,5.810,149.146
C07982=1175.670,-35.305,-43.808,179.625,5.810,149.145
C07983=1175.665,-35.056,-43.821,179.627,5.811,149.144
C07984=1175.660,-34.806,-43.833,179.630,5.811,149.144
C07985=1175.655,-34.556,-43.844,179.632,5.812,149.143
C07986=1175.650,-34.307,-43.857,179.635,5.813,149.143
C07987=1175.644,-34.057,-43.869,179.637,5.812,149.142
C07988=1175.639,-33.808,-43.881,179.639,5.813,149.141
C07989=1175.634,-33.558,-43.893,179.642,5.813,149.141
C07990=1175.629,-33.309,-43.906,179.644,5.814,149.140
C07991=1175.623,-33.059,-43.918,179.646,5.815,149.140
C07992=1175.618,-32.809,-43.930,179.649,5.815,149.139
C07993=1175.613,-32.560,-43.941,179.651,5.815,149.138
C07994=1175.608,-32.310,-43.953,179.653,5.816,149.138
C07995=1175.603,-32.060,-43.966,179.656,5.816,149.137
C07996=1175.597,-31.811,-43.978,179.659,5.817,149.136
C07997=1175.592,-31.561,-43.990,179.661,5.817,149.136
C07998=1175.588,-31.311,-44.003,179.664,5.818,149.135
C07999=1175.582,-31.061,-44.015,179.666,5.818,149.134
C08000=1175.577,-30.812,-44.028,179.668,5.818,149.134
C08001=1175.572,-30.562,-44.040,179.670,5.819,149.133
C08002=1175.567,-30.313,-44.052,179.673,5.819,149.133
C08003=1175.561,-30.063,-44.064,179.675,5.820,149.132
C08004=1175.556,-29.813,-44.077,179.678,5.820,149.131
C08005=1175.551,-29.564,-44.089,179.681,5.821,149.131
C08006=1175.546,-29.314,-44.101,179.683,5.822,149.130
C08007=1175.540,-29.065,-44.114,179.685,5.821,149.130
C08008=1175.536,-28.814,-44.126,179.688,5.822,149.129
C08009=1175.530,-28.565,-44.139,179.690,5.823,149.128
C08010=1175.525,-28.315,-44.151,179.692,5.823,149.128
C08011=1175.520,-28.066,-44.163,179.695,5.823,149.127
C08012=1175.515,-27.816,-44.176,179.697,5.824,149.126
C08013=1175.509,-27.566,-44.188,179.700,5.825,149.126
C08014=1175.504,-27.317,-44.200,179.702,5.826,149.125
C08015=1175.499,-27.068,-44.213,179.704,5.825,149.125
C08016=1175.494,-26.817,-44.225,179.707,5.826,149.124
C08017=1175.489,-26.568,-44.238,179.709,5.826,149.123
C08018=1175.484,-26.318,-44.250,179.712,5.827,149.123
C08019=1175.479,-26.069,-44.262,179.714,5.827,149.122
C08020=1175.473,-25.819,-44.275,179.716,5.828,149.122
C08021=1175.468,-25.570,-44.288,179.719,5.829,149.121
C08022=1175.464,-25.319,-44.300,179.722,5.829,149.120
C08023=1175.458,-25.070,-44.312,179.723,5.829,149.120
C08024=1175.453,-24.821,-44.325,179.726,5.829,149.119
C08025=1175.448,-24.571,-44.338,179.729,5.830,149.118
C08026=1175.443,-24.321,-44.349,179.731,5.831,149.118
C08027=1175.437,-24.051,-44.364,179.734,5.831,149.117
C08028=1175.432,-23.782,-44.377,179.736,5.832,149.116
C08029=1175.426,-23.513,-44.391,179.739,5.832,149.116
C08030=1175.420,-23.242,-44.404,179.742,5.833,149.115
C08031=1175.415,-22.993,-44.417,179.744,5.833,149.114
C08032=1175.410,-22.743,-44.429,179.746,5.834,149.114
C08033=1175.406,-22.493,-44.442,179.749,5.834,149.113
C08034=1175.400,-22.243,-44.454,179.751,5.835,149.113
C08035=1175.395,-21.994,-44.467,179.754,5.835,149.112
C08036=1175.390,-21.745,-44.480,179.757,5.836,149.111
C08037=1175.384,-21.495,-44.493,179.759,5.837,149.111
C08038=1175.379,-21.245,-44.506,179.761,5.836,149.110
C08039=1175.374,-20.996,-44.518,179.763,5.837,149.109
C08040=1175.369,-20.746,-44.530,179.766,5.838,149.109
C08041=1175.364,-20.496,-44.543,179.768,5.838,149.108
C08042=1175.359,-20.246,-44.556,179.771,5.839,149.108
C08043=1175.353,-19.997,-44.569,179.773,5.839,149.107
C08044=1175.348,-19.748,-44.582,179.776,5.840,149.106
C08045=1175.343,-19.498,-44.594,179.778,5.840,149.106
C08046=1175.339,-19.248,-44.607,179.781,5.841,149.105
C08047=1175.334,-18.999,-44.620,179.783,5.842,149.105
C08048=1175.328,-18.749,-44.633,179.786,5.842,149.104
C08049=1175.322,-18.499,-44.645,179.788,5.842,149.103
C08050=1175.318,-18.249,-44.658,179.790,5.842,149.103
C08051=1175.313,-18.000,-44.670,179.793,5.843,149.102
C08052=1175.307,-17.750,-44.684,179.795,5.844,149.102
C08053=1175.302,-17.501,-44.696,179.798,5.844,149.101
C08054=1175.297,-17.251,-44.709,179.800,5.845,149.100
C08055=1175.292,-17.002,-44.722,179.803,5.846,149.100
C08056=1175.286,-16.752,-44.735,179.805,5.846,149.099
C08057=1175.282,-16.502,-44.748,179.808,5.846,149.098
C08058=1175.276,-16.253,-44.760,179.810,5.847,149.098
C08059=1175.271,-16.003,-44.773,179.813,5.848,149.097
C08060=1175.266,-15.753,-44.787,179.815,5.848,149.096
C08061=1175.261,-15.504,-44.799,179.818,5.849,149.096
C08062=1175.256,-15.254,-44.812,179.820,5.849,149.095
C08063=1175.251,-15.004,-44.825,179.822,5.849,149.095
C08064=1175.245,-14.755,-44.838,179.824,5.850,149.094
C08065=1175.240,-14.505,-44.851,179.827,5.850,149.093
C08066=1175.236,-14.255,-44.864,179.830,5.851,149.093
C08067=1175.230,-14.006,-44.877,179.832,5.852,149.092
C08068=1175.225,-13.757,-44.890,179.835,5.852,149.092
C08069=1175.221,-13.507,-44.903,179.837,5.853,149.091
C08070=1175.215,-13.257,-44.916,179.839,5.853,149.090
C08071=1175.210,-13.008,-44.929,179.842,5.854,149.090
C08072=1175.205,-12.758,-44.942,179.845,5.854,149.089
C08073=1175.199,-12.509,-44.955,179.847,5.855,149.089
C08074=1175.194,-12.259,-44.968,179.850,5.856,149.088
C08075=1175.189,-12.009,-44.981,179.852,5.856,149.087
C08076=1175.184,-11.760,-44.994,179.854,5.857,149.087
C08077=1175.179,-11.511,-45.007,179.857,5.857,149.086
C08078=1175.174,-11.261,-45.021,179.859,5.858,149.086
C08079=1175.169,-11.011,-45.033,179.861,5.858,149.085
C08080=1175.164,-10.761,-45.046,179.864,5.858,149.084
C08081=1175.158,-10.512,-45.059,179.866,5.859,149.084
C08082=1175.153,-10.262,-45.072,179.869,5.860,149.083
C08083=1175.148,-10.013,-45.086,179.871,5.860,149.082
C08084=1175.143,-9.763,-45.099,179.874,5.861,149.082
C08085=1175.138,-9.513,-45.112,179.876,5.861,149.081
C08086=1175.133,-9.264,-45.125,179.879,5.862,149.081
C08087=1175.128,-9.015,-45.138,179.881,5.863,149.080
C08088=1175.122,-8.765,-45.152,179.884,5.863,149.079
C08089=1175.117,-8.515,-45.165,179.886,5.863,149.079
C08090=1175.112,-8.265,-45.178,179.889,5.864,149.078
C08091=1175.107,-8.016,-45.191,179.891,5.865,149.078
C08092=1175.103,-7.766,-45.204,179.894,5.865,149.077
C08093=1175.097,-7.517,-45.218,179.896,5.866,149.076
C08094=1175.092,-7.267,-45.231,179.899,5.867,149.076
C08095=1175.087,-7.018,-45.244,179.901,5.867,149.075
C08096=1175.082,-6.768,-45.257,179.904,5.868,149.075
C08097=1175.076,-6.518,-45.271,179.906,5.868,149.074
C08098=1175.072,-6.269,-45.284,179.909,5.869,149.073
C08099=1175.066,-6.019,-45.298,179.911,5.870,149.073
C08100=1175.061,-5.770,-45.310,179.914,5.870,149.072
C08101=1175.056,-5.520,-45.324,179.916,5.870,149.071
C08102=1175.051,-5.271,-45.337,179.918,5.871,149.071
C08103=1175.046,-5.020,-45.351,179.921,5.872,149.070
C08104=1175.041,-4.771,-45.364,179.924,5.872,149.069
C08105=1175.036,-4.521,-45.377,179.926,5.873,149.069
C08106=1175.030,-4.272,-45.391,179.929,5.874,149.068
C08107=1175.026,-4.022,-45.404,179.931,5.874,149.068
C08108=1175.020,-3.772,-45.418,179.933,5.875,149.067
C08109=1175.016,-3.523,-45.431,179.936,5.875,149.066
C08110=1175.010,-3.273,-45.444,179.938,5.876,149.066
C08111=1175.006,-3.024,-45.458,179.941,5.877,149.065
C08112=1175.000,-2.774,-45.471,179.944,5.877,149.065
C08113=1174.994,-2.524,-45.485,179.946,5.878,149.064
C08114=1174.990,-2.275,-45.498,179.948,5.878,149.063
C08115=1174.984,-2.025,-45.512,179.951,5.879,149.063
C08116=1174.980,-1.776,-45.525,179.953,5.880,149.062
C08117=1174.974,-1.526,-45.539,179.956,5.880,149.062
C08118=1174.969,-1.277,-45.552,179.959,5.881,149.061
C08119=1174.964,-1.027,-45.565,179.961,5.881,149.060
C08120=1174.959,-0.778,-45.579,179.963,5.882,149.060
C08121=1174.954,-0.528,-45.592,179.966,5.882,149.059
C08122=1174.949,-0.279,-45.606,179.968,5.883,149.059
C08123=1174.943,-0.029,-45.620,179.971,5.884,149.058
C08124=1174.939,0.221,-45.633,179.974,5.884,149.057
C08125=1174.933,0.470,-45.647,179.976,5.885,149.057
C08126=1174.928,0.720,-45.661,179.978,5.885,149.056
C08127=1174.923,0.969,-45.674,179.981,5.886,149.055
C08128=1174.918,1.219,-45.688,179.983,5.887,149.055
C08129=1174.913,1.468,-45.702,179.986,5.887,149.054
C08130=1174.908,1.718,-45.715,179.988,5.888,149.054
C08131=1174.903,1.988,-45.730,179.991,5.888,149.053
C08132=1174.897,2.256,-45.744,179.993,5.889,149.052
C08133=1174.891,2.526,-45.759,179.996,5.889,149.052
C08134=1174.886,2.795,-45.774,179.999,5.891,149.051
C08135=1174.881,3.045,-45.787,-179.998,5.891,149.050
C08136=1174.876,3.294,-45.801,-179.996,5.892,149.050
C08137=1174.871,3.544,-45.815,-179.993,5.892,149.049
C08138=1174.865,3.793,-45.829,-179.991,5.893,149.049
C08139=1174.861,4.043,-45.842,-179.988,5.894,149.048
C08140=1174.856,4.293,-45.857,-179.986,5.894,149.047
C08141=1174.850,4.542,-45.870,-179.984,5.895,149.047
C08142=1174.845,4.792,-45.884,-179.981,5.896,149.046
C08143=1174.841,5.041,-45.898,-179.978,5.896,149.046
C08144=1174.835,5.291,-45.911,-179.976,5.897,149.045
C08145=1174.830,5.541,-45.925,-179.974,5.897,149.044
C08146=1174.824,5.790,-45.939,-179.971,5.898,149.044
C08147=1174.820,6.039,-45.953,-179.969,5.899,149.043
C08148=1174.815,6.289,-45.966,-179.966,5.899,149.043
C08149=1174.809,6.538,-45.980,-179.963,5.900,149.042
C08150=1174.804,6.788,-45.995,-179.961,5.900,149.041
C08151=1174.799,7.038,-46.009,-179.959,5.901,149.041
C08152=1174.794,7.287,-46.021,-179.956,5.901,149.040
C08153=1174.789,7.537,-46.036,-179.954,5.902,149.040
C08154=1174.784,7.787,-46.050,-179.951,5.903,149.039
C08155=1174.779,8.036,-46.064,-179.949,5.903,149.038
C08156=1174.774,8.285,-46.078,-179.946,5.905,149.038
C08157=1174.769,8.536,-46.092,-179.943,5.905,149.037
C08158=1174.764,8.785,-46.105,-179.941,5.906,149.037
C08159=1174.759,9.034,-46.119,-179.938,5.907,149.036
C08160=1174.754,9.284,-46.134,-179.936,5.907,149.035
C08161=1174.749,9.533,-46.148,-179.933,5.908,149.035
C08162=1174.743,9.782,-46.162,-179.931,5.908,149.034
C08163=1174.738,10.033,-46.175,-179.928,5.909,149.033
C08164=1174.733,10.283,-46.190,-179.926,5.910,149.033
C08165=1174.728,10.532,-46.204,-179.923,5.910,149.032
C08166=1174.723,10.781,-46.217,-179.921,5.911,149.032
C08167=1174.718,11.031,-46.232,-179.918,5.911,149.031
C08168=1174.713,11.280,-46.246,-179.916,5.912,149.030
C08169=1174.708,11.529,-46.260,-179.914,5.913,149.030
C08170=1174.703,11.779,-46.274,-179.911,5.913,149.029
C08171=1174.698,12.029,-46.288,-179.908,5.914,149.029
C08172=1174.693,12.278,-46.303,-179.906,5.915,149.028
C08173=1174.687,12.528,-46.316,-179.903,5.916,149.027
C08174=1174.682,12.778,-46.330,-179.900,5.916,149.027
C08175=1174.677,13.028,-46.344,-179.898,5.917,149.026
C08176=1174.672,13.277,-46.359,-179.895,5.918,149.026
C08177=1174.667,13.526,-46.373,-179.893,5.918,149.025
C08178=1174.662,13.776,-46.387,-179.891,5.919,149.025
C08179=1174.657,14.026,-46.401,-179.888,5.919,149.024
C08180=1174.652,14.275,-46.415,-179.886,5.920,149.023
C08181=1174.647,14.525,-46.430,-179.883,5.921,149.023
C08182=1174.641,14.774,-46.444,-179.880,5.922,149.022
C08183=1174.636,15.024,-46.458,-179.878,5.923,149.022
C08184=1174.631,15.274,-46.472,-179.875,5.923,149.021
C08185=1174.627,15.523,-46.487,-179.873,5.924,149.020
C08186=1174.621,15.772,-46.501,-179.870,5.925,149.020
C08187=1174.616,16.021,-46.515,-179.868,5.925,149.019
C08188=1174.611,16.271,-46.530,-179.865,5.926,149.018
C08189=1174.606,16.521,-46.544,-179.863,5.926,149.018
C08190=1174.601,16.770,-46.558,-179.860,5.927,149.017
C08191=1174.596,17.020,-46.572,-179.858,5.928,149.017
C08192=1174.591,17.269,-46.586,-179.855,5.929,149.016
C08193=1174.586,17.519,-46.601,-179.852,5.930,149.015
C08194=1174.581,17.769,-46.615,-179.850,5.930,149.015
C08195=1174.576,18.018,-46.629,-179.847,5.931,149.014
C08196=1174.571,18.267,-46.644,-179.845,5.931,149.014
C08197=1174.566,18.517,-46.658,-179.843,5.932,149.013
C08198=1174.561,18.766,-46.672,-179.840,5.933,149.012
C08199=1174.556,19.016,-46.687,-179.838,5.934,149.012
C08200=1174.550,19.266,-46.701,-179.835,5.934,149.011
C08201=1174.545,19.516,-46.716,-179.832,5.935,149.011
C08202=1174.541,19.765,-46.731,-179.830,5.936,149.010
C08203=1174.536,20.014,-46.745,-179.827,5.937,149.009
C08204=1174.531,20.264,-46.759,-179.824,5.937,149.009
C08205=1174.526,20.514,-46.774,-179.822,5.938,149.008
C08206=1174.521,20.762,-46.788,-179.820,5.938,149.008
C08207=1174.516,21.012,-46.802,-179.817,5.939,149.007
C08208=1174.510,21.262,-46.817,-179.815,5.940,149.007
C08209=1174.505,21.512,-46.832,-179.812,5.941,149.006
C08210=1174.500,21.761,-46.847,-179.809,5.942,149.005
C08211=1174.495,22.010,-46.861,-179.807,5.942,149.005
C08212=1174.490,22.260,-46.875,-179.804,5.943,149.004
C08213=1174.485,22.510,-46.889,-179.802,5.944,149.004
C08214=1174.480,22.759,-46.905,-179.799,5.944,149.003
C08215=1174.475,23.009,-46.919,-179.797,5.945,149.002
C08216=1174.469,23.258,-46.933,-179.794,5.946,149.002
C08217=1174.465,23.507,-46.948,-179.791,5.947,149.001
C08218=1174.460,23.757,-46.962,-179.789,5.948,149.001
C08219=1174.454,24.007,-46.977,-179.786,5.948,149.000
C08220=1174.450,24.256,-46.992,-179.784,5.949,149.000
C08221=1174.445,24.506,-47.007,-179.782,5.950,148.999
C08222=1174.440,24.755,-47.021,-179.779,5.950,148.998
C08223=1174.435,25.004,-47.036,-179.776,5.952,148.998
C08224=1174.429,25.254,-47.051,-179.774,5.952,148.997
C08225=1174.425,25.503,-47.066,-179.771,5.953,148.996
C08226=1174.420,25.753,-47.080,-179.769,5.953,148.996
C08227=1174.414,26.003,-47.095,-179.766,5.954,148.995
C08228=1174.409,26.252,-47.110,-179.764,5.955,148.995
C08229=1174.404,26.502,-47.124,-179.761,5.956,148.994
C08230=1174.400,26.751,-47.139,-179.758,5.957,148.993
C08231=1174.394,27.001,-47.154,-179.756,5.957,148.993
C08232=1174.389,27.250,-47.169,-179.753,5.958,148.992
C08233=1174.384,27.500,-47.183,-179.751,5.959,148.992
C08234=1174.379,27.750,-47.198,-179.748,5.959,148.991
C08235=1174.374,28.018,-47.215,-179.745,5.961,148.990
C08236=1174.369,28.287,-47.230,-179.743,5.961,148.990
C08237=1174.363,28.556,-47.247,-179.740,5.962,148.989
C08238=1174.358,28.825,-47.262,-179.737,5.963,148.989
C08239=1174.352,29.075,-47.277,-179.735,5.964,148.988
C08240=1174.347,29.324,-47.292,-179.732,5.964,148.987
C08241=1174.343,29.574,-47.306,-179.730,5.965,148.987
C08242=1174.337,29.823,-47.322,-179.727,5.966,148.986
C08243=1174.332,30.073,-47.336,-179.724,5.967,148.986
C08244=1174.328,30.322,-47.351,-179.722,5.968,148.985
C08245=1174.322,30.571,-47.367,-179.719,5.968,148.984
C08246=1174.317,30.821,-47.381,-179.717,5.969,148.984
C08247=1174.313,31.070,-47.396,-179.714,5.970,148.983
C08248=1174.307,31.320,-47.411,-179.711,5.971,148.983
C08249=1174.302,31.569,-47.426,-179.709,5.972,148.982
C08250=1174.297,31.819,-47.442,-179.706,5.972,148.981
C08251=1174.292,32.068,-47.456,-179.704,5.973,148.981
C08252=1174.287,32.317,-47.471,-179.701,5.974,148.980
C08253=1174.282,32.567,-47.486,-179.699,5.974,148.980
C08254=1174.277,32.816,-47.501,-179.696,5.976,148.979
C08255=1174.271,33.066,-47.516,-179.693,5.976,148.979
C08256=1174.267,33.316,-47.531,-179.691,5.977,148.978
C08257=1174.262,33.566,-47.547,-179.689,5.978,148.977
C08258=1174.257,33.815,-47.562,-179.686,5.978,148.977
C08259=1174.251,34.065,-47.576,-179.683,5.980,148.976
C08260=1174.247,34.314,-47.591,-179.681,5.980,148.976
C08261=1174.241,34.563,-47.607,-179.678,5.981,148.975
C08262=1174.237,34.812,-47.622,-179.676,5.982,148.974
C08263=1174.231,35.062,-47.637,-179.674,5.982,148.974
C08264=1174.226,35.312,-47.652,-179.670,5.984,148.973
C08265=1174.221,35.561,-47.667,-179.668,5.984,148.973
C08266=1174.217,35.811,-47.683,-179.666,5.985,148.972
C08267=1174.211,36.061,-47.698,-179.663,5.986,148.972
C08268=1174.207,36.310,-47.713,-179.660,5.987,148.971
C08269=1174.201,36.559,-47.728,-179.657,5.988,148.970
C08270=1174.197,36.808,-47.743,-179.655,5.989,148.970
C08271=1174.191,37.058,-47.759,-179.653,5.989,148.969
C08272=1174.186,37.307,-47.773,-179.650,5.990,148.969
C08273=1174.181,37.558,-47.789,-179.647,5.991,148.968
C08274=1174.177,37.807,-47.804,-179.645,5.992,148.968
C08275=1174.171,38.056,-47.820,-179.642,5.993,148.967
C08276=1174.166,38.305,-47.835,-179.640,5.993,148.966
C08277=1174.161,38.555,-47.850,-179.637,5.994,148.966
C08278=1174.156,38.805,-47.865,-179.634,5.995,148.965
C08279=1174.152,39.054,-47.880,-179.632,5.996,148.965
C08280=1174.146,39.304,-47.896,-179.630,5.997,148.964
C08281=1174.142,39.553,-47.911,-179.626,5.998,148.963
C08282=1174.136,39.802,-47.927,-179.624,5.999,148.963
C08283=1174.131,40.052,-47.942,-179.622,5.999,148.962
C08284=1174.127,40.301,-47.958,-179.619,6.000,148.962
C08285=1174.121,40.551,-47.973,-179.616,6.001,148.961
C08286=1174.116,40.800,-47.989,-179.614,6.002,148.961
C08287=1174.111,41.049,-48.004,-179.611,6.003,148.960
C08288=1174.106,41.299,-48.019,-179.609,6.003,148.959
C08289=1174.101,41.549,-48.035,-179.606,6.004,148.959
C08290=1174.096,41.799,-48.050,-179.603,6.005,148.958
C08291=1174.091,42.048,-48.065,-179.601,6.006,148.958
C08292=1174.085,42.297,-48.081,-179.599,6.007,148.957
C08293=1174.081,42.547,-48.096,-179.596,6.007,148.957
C08294=1174.076,42.797,-48.112,-179.593,6.009,148.956
C08295=1174.071,43.046,-48.127,-179.591,6.009,148.955
C08296=1174.066,43.295,-48.142,-179.588,6.010,148.955
C08297=1174.061,43.545,-48.158,-179.585,6.012,148.954
C08298=1174.056,43.794,-48.175,-179.583,6.012,148.954
C08299=1174.051,44.043,-48.190,-179.580,6.013,148.953
C08300=1174.046,44.292,-48.205,-179.578,6.014,148.953
C08301=1174.041,44.543,-48.221,-179.575,6.015,148.952
C08302=1174.036,44.792,-48.237,-179.572,6.016,148.951
C08303=1174.031,45.041,-48.252,-179.570,6.016,148.951
C08304=1174.026,45.290,-48.267,-179.568,6.017,148.950
C08305=1174.021,45.541,-48.283,-179.564,6.018,148.950
C08306=1174.016,45.790,-48.299,-179.562,6.019,148.949
C08307=1174.011,46.039,-48.314,-179.560,6.020,148.949
C08308=1174.006,46.289,-48.330,-179.557,6.021,148.948
C08309=1174.001,46.538,-48.346,-179.554,6.022,148.947
C08310=1173.996,46.787,-48.362,-179.552,6.023,148.947
C08311=1173.992,47.037,-48.377,-179.549,6.023,148.946
C08312=1173.986,47.286,-48.393,-179.546,6.025,148.946
C08313=1173.981,47.536,-48.408,-179.544,6.025,148.945
C08314=1173.976,47.786,-48.424,-179.541,6.026,148.945
C08315=1173.971,48.035,-48.440,-179.539,6.027,148.944
C08316=1173.966,48.284,-48.456,-179.536,6.028,148.943
C08317=1173.962,48.534,-48.471,-179.534,6.029,148.943
C08318=1173.956,48.783,-48.487,-179.531,6.030,148.942
C08319=1173.951,49.032,-48.503,-179.528,6.031,148.942
C08320=1173.946,49.282,-48.519,-179.526,6.032,148.941
C08321=1173.941,49.532,-48.535,-179.523,6.032,148.941
C08322=1173.936,49.781,-48.550,-179.520,6.034,148.940
C08323=1173.932,50.030,-48.566,-179.518,6.034,148.939
C08324=1173.926,50.280,-48.582,-179.516,6.035,148.939
C08325=1173.921,50.529,-48.598,-179.513,6.036,148.938
C08326=1173.916,50.779,-48.614,-179.510,6.037,148.938
C08327=1173.911,51.028,-48.630,-179.508,6.038,148.937
C08328=1173.906,51.278,-48.646,-179.505,6.039,148.937
C08329=1173.901,51.527,-48.661,-179.502,6.040,148.936
C08330=1173.896,51.776,-48.678,-179.500,6.041,148.935
C08331=1173.891,52.026,-48.694,-179.497,6.041,148.935
C08332=1173.887,52.275,-48.709,-179.494,6.043,148.934
C08333=1173.882,52.525,-48.725,-179.492,6.044,148.934
C08334=1173.877,52.774,-48.741,-179.489,6.044,148.933
C08335=1173.872,53.023,-48.757,-179.487,6.046,148.933
C08336=1173.867,53.273,-48.773,-179.484,6.046,148.932
C08337=1173.861,53.523,-48.789,-179.482,6.047,148.932
C08338=1173.857,53.772,-48.805,-179.479,6.049,148.931
C08339=1173.851,54.041,-48.822,-179.476,6.049,148.930
C08340=1173.846,54.309,-48.839,-179.473,6.051,148.930
C08341=1173.840,54.578,-48.857,-179.471,6.051,148.929
C08342=1173.836,54.846,-48.875,-179.467,6.053,148.929
C08343=1173.830,55.095,-48.890,-179.465,6.053,148.928
C08344=1173.826,55.345,-48.907,-179.463,6.054,148.927
C08345=1173.820,55.594,-48.922,-179.460,6.056,148.927
C08346=1173.816,55.844,-48.938,-179.457,6.056,148.926
C08347=1173.811,56.093,-48.955,-179.455,6.057,148.926
C08348=1173.805,56.343,-48.970,-179.452,6.058,148.925
C08349=1173.801,56.592,-48.987,-179.449,6.059,148.925
C08350=1173.795,56.842,-49.003,-179.447,6.060,148.924
C08351=1173.790,57.091,-49.020,-179.444,6.061,148.923
C08352=1173.785,57.340,-49.036,-179.442,6.062,148.923
C08353=1173.780,57.590,-49.052,-179.439,6.062,148.922
C08354=1173.775,57.839,-49.068,-179.436,6.064,148.922
C08355=1173.770,58.089,-49.084,-179.434,6.065,148.921
C08356=1173.765,58.338,-49.101,-179.432,6.066,148.921
C08357=1173.760,58.588,-49.117,-179.428,6.067,148.920
C08358=1173.755,58.837,-49.133,-179.426,6.068,148.920
C08359=1173.751,59.086,-49.150,-179.424,6.068,148.919
C08360=1173.745,59.336,-49.165,-179.421,6.070,148.919
C08361=1173.741,59.585,-49.182,-179.418,6.070,148.918
C08362=1173.735,59.835,-49.198,-179.416,6.071,148.918
C08363=1173.730,60.084,-49.215,-179.413,6.073,148.917
C08364=1173.726,60.334,-49.231,-179.411,6.073,148.916
C08365=1173.721,60.583,-49.247,-179.408,6.075,148.916
C08366=1173.716,60.833,-49.264,-179.405,6.076,148.915
C08367=1173.711,61.081,-49.280,-179.403,6.076,148.915
C08368=1173.706,61.332,-49.296,-179.399,6.078,148.914
C08369=1173.700,61.581,-49.313,-179.397,6.078,148.914
C08370=1173.696,61.830,-49.329,-179.395,6.079,148.913
C08371=1173.691,62.079,-49.346,-179.392,6.081,148.912
C08372=1173.686,62.329,-49.362,-179.389,6.081,148.912
C08373=1173.682,62.579,-49.378,-179.387,6.083,148.911
C08374=1173.676,62.827,-49.395,-179.384,6.083,148.911
C08375=1173.671,63.077,-49.412,-179.382,6.084,148.910
C08376=1173.666,63.327,-49.428,-179.379,6.086,148.910
C08377=1173.661,63.576,-49.444,-179.376,6.086,148.909
C08378=1173.657,63.825,-49.461,-179.374,6.087,148.908
C08379=1173.651,64.075,-49.478,-179.371,6.089,148.908
C08380=1173.647,64.324,-49.494,-179.368,6.089,148.907
C08381=1173.641,64.573,-49.510,-179.366,6.091,148.907
C08382=1173.637,64.823,-49.527,-179.363,6.091,148.906
C08383=1173.632,65.072,-49.543,-179.361,6.092,148.906
C08384=1173.626,65.322,-49.560,-179.358,6.094,148.905
C08385=1173.622,65.571,-49.577,-179.356,6.094,148.905
C08386=1173.617,65.821,-49.594,-179.352,6.096,148.904
C08387=1173.611,66.070,-49.610,-179.350,6.097,148.904
C08388=1173.607,66.320,-49.626,-179.348,6.097,148.903
C08389=1173.602,66.568,-49.643,-179.345,6.099,148.903
C08390=1173.597,66.818,-49.659,-179.342,6.099,148.902
C08391=1173.592,67.068,-49.677,-179.339,6.101,148.902
C08392=1173.587,67.317,-49.693,-179.337,6.102,148.901
C08393=1173.583,67.566,-49.710,-179.335,6.102,148.900
C08394=1173.577,67.816,-49.727,-179.331,6.104,148.900
C08395=1173.572,68.065,-49.743,-179.329,6.105,148.899
C08396=1173.568,68.314,-49.760,-179.326,6.106,148.899
C08397=1173.563,68.564,-49.777,-179.324,6.107,148.898
C08398=1173.558,68.813,-49.794,-179.321,6.108,148.898
C08399=1173.553,69.062,-49.810,-179.319,6.109,148.897
C08400=1173.548,69.312,-49.827,-179.316,6.110,148.897
C08401=1173.543,69.561,-49.844,-179.313,6.111,148.896
C08402=1173.537,69.811,-49.861,-179.311,6.112,148.896
C08403=1173.533,70.060,-49.878,-179.308,6.114,148.895
C08404=1173.528,70.309,-49.894,-179.306,6.114,148.895
C08405=1173.523,70.559,-49.911,-179.303,6.116,148.894
C08406=1173.518,70.808,-49.928,-179.300,6.117,148.893
C08407=1173.513,71.058,-49.945,-179.298,6.117,148.893
C08408=1173.508,71.307,-49.962,-179.295,6.119,148.892
C08409=1173.503,71.556,-49.978,-179.292,6.119,148.892
C08410=1173.498,71.806,-49.995,-179.290,6.121,148.891
C08411=1173.494,72.055,-50.012,-179.287,6.122,148.891
C08412=1173.489,72.305,-50.029,-179.284,6.123,148.890
C08413=1173.483,72.554,-50.046,-179.282,6.124,148.890
C08414=1173.478,72.804,-50.063,-179.280,6.125,148.889
C08415=1173.474,73.053,-50.080,-179.276,6.126,148.888
C08416=1173.469,73.302,-50.097,-179.274,6.127,148.888
C08417=1173.464,73.551,-50.114,-179.271,6.128,148.887
C08418=1173.459,73.801,-50.131,-179.269,6.129,148.887
C08419=1173.454,74.051,-50.148,-179.266,6.130,148.886
C08420=1173.449,74.300,-50.165,-179.263,6.131,148.886
C08421=1173.444,74.548,-50.182,-179.261,6.133,148.885
C08422=1173.439,74.798,-50.199,-179.258,6.134,148.885
C08423=1173.434,75.048,-50.216,-179.256,6.134,148.884
C08424=1173.429,75.298,-50.233,-179.253,6.136,148.884
C08425=1173.425,75.546,-50.251,-179.251,6.137,148.883
C08426=1173.419,75.796,-50.267,-179.247,6.138,148.883
C08427=1173.415,76.045,-50.284,-179.245,6.139,148.882
C08428=1173.409,76.295,-50.301,-179.242,6.140,148.881
C08429=1173.405,76.544,-50.319,-179.240,6.141,148.881
C08430=1173.400,76.793,-50.336,-179.237,6.142,148.880
C08431=1173.396,77.043,-50.353,-179.235,6.143,148.880
C08432=1173.390,77.292,-50.370,-179.232,6.145,148.880
C08433=1173.385,77.541,-50.388,-179.229,6.146,148.879
C08434=1173.380,77.791,-50.404,-179.226,6.147,148.878
C08435=1173.375,78.040,-50.422,-179.224,6.148,148.878
C08436=1173.371,78.289,-50.439,-179.221,6.149,148.877
C08437=1173.366,78.539,-50.456,-179.218,6.150,148.877
C08438=1173.360,78.788,-50.473,-179.216,6.152,148.876
C08439=1173.356,79.037,-50.490,-179.213,6.152,148.876
C08440=1173.351,79.287,-50.508,-179.210,6.154,148.875
C08441=1173.346,79.536,-50.526,-179.208,6.154,148.875
C08442=1173.341,79.786,-50.542,-179.206,6.155,148.874
C08443=1173.336,80.054,-50.561,-179.202,6.157,148.874
C08444=1173.330,80.323,-50.579,-179.200,6.158,148.873
C08445=1173.325,80.591,-50.598,-179.196,6.160,148.872
C08446=1173.320,80.859,-50.617,-179.194,6.161,148.872
C08447=1173.315,81.109,-50.635,-179.191,6.162,148.871
C08448=1173.309,81.358,-50.652,-179.189,6.163,148.871
C08449=1173.305,81.607,-50.668,-179.186,6.164,148.870
C08450=1173.300,81.856,-50.686,-179.184,6.165,148.870
C08451=1173.295,82.106,-50.704,-179.180,6.166,148.869
C08452=1173.291,82.355,-50.721,-179.178,6.167,148.869
C08453=1173.285,82.605,-50.738,-179.176,6.169,148.868
C08454=1173.280,82.854,-50.756,-179.173,6.170,148.868
C08455=1173.275,83.104,-50.774,-179.170,6.171,148.867
C08456=1173.271,83.353,-50.791,-179.168,6.172,148.867
C08457=1173.266,83.602,-50.809,-179.165,6.173,148.866
C08458=1173.261,83.852,-50.826,-179.162,6.174,148.866
C08459=1173.256,84.101,-50.844,-179.159,6.176,148.865
C08460=1173.251,84.350,-50.861,-179.157,6.177,148.865
C08461=1173.247,84.599,-50.879,-179.154,6.178,148.864
C08462=1173.241,84.849,-50.896,-179.152,6.179,148.864
C08463=1173.236,85.098,-50.914,-179.149,6.180,148.863
C08464=1173.232,85.348,-50.932,-179.147,6.181,148.863
C08465=1173.227,85.597,-50.949,-179.143,6.182,148.862
C08466=1173.222,85.846,-50.967,-179.141,6.183,148.861
C08467=1173.217,86.095,-50.984,-179.139,6.185,148.861
C08468=1173.211,86.345,-51.002,-179.135,6.186,148.860
C08469=1173.206,86.594,-51.020,-179.133,6.187,148.860
C08470=1173.202,86.843,-51.037,-179.130,6.189,148.859
C08471=1173.197,87.092,-51.054,-179.128,6.190,148.859
C08472=1173.192,87.342,-51.072,-179.125,6.191,148.859
C08473=1173.187,87.591,-51.090,-179.123,6.192,148.858
C08474=1173.183,87.841,-51.108,-179.120,6.193,148.857
C08475=1173.178,88.090,-51.126,-179.117,6.194,148.857
C08476=1173.173,88.340,-51.144,-179.114,6.196,148.856
C08477=1173.169,88.588,-51.161,-179.112,6.197,148.856
C08478=1173.163,88.838,-51.178,-179.109,6.198,148.855
C08479=1173.159,89.087,-51.196,-179.107,6.199,148.855
C08480=1173.154,89.337,-51.214,-179.104,6.200,148.854
C08481=1173.149,89.586,-51.232,-179.101,6.202,148.854
C08482=1173.143,89.836,-51.250,-179.099,6.203,148.853
C08483=1173.139,90.085,-51.268,-179.096,6.204,148.853
C08484=1173.134,90.334,-51.286,-179.094,6.205,148.852
C08485=1173.129,90.583,-51.304,-179.090,6.206,148.852
C08486=1173.124,90.832,-51.322,-179.088,6.207,148.851
C08487=1173.119,91.082,-51.339,-179.085,6.209,148.851
C08488=1173.114,91.331,-51.357,-179.082,6.210,148.850
C08489=1173.109,91.580,-51.375,-179.080,6.211,148.850
C08490=1173.104,91.830,-51.393,-179.077,6.213,148.849
C08491=1173.099,92.079,-51.411,-179.075,6.213,148.849
C08492=1173.095,92.329,-51.429,-179.072,6.215,148.848
C08493=1173.090,92.578,-51.447,-179.069,6.216,148.848
C08494=1173.085,92.827,-51.465,-179.067,6.217,148.847
C08495=1173.080,93.076,-51.483,-179.065,6.218,148.847
C08496=1173.075,93.326,-51.500,-179.061,6.220,148.846
C08497=1173.070,93.575,-51.518,-179.059,6.221,148.846
C08498=1173.065,93.824,-51.536,-179.056,6.222,148.845
C08499=1173.060,94.073,-51.554,-179.053,6.224,148.845
C08500=1173.056,94.323,-51.573,-179.051,6.225,148.844
C08501=1173.051,94.573,-51.591,-179.048,6.226,148.844
C08502=1173.046,94.822,-51.609,-179.045,6.228,148.843
C08503=1173.041,95.071,-51.627,-179.043,6.229,148.843
C08504=1173.036,95.320,-51.645,-179.040,6.230,148.842
C08505=1173.031,95.569,-51.662,-179.038,6.231,148.842
C08506=1173.026,95.818,-51.680,-179.035,6.232,148.841
C08507=1173.022,96.068,-51.699,-179.032,6.234,148.841
C08508=1173.017,96.317,-51.717,-179.030,6.235,148.840
C08509=1173.012,96.567,-51.735,-179.027,6.236,148.840
C08510=1173.006,96.816,-51.753,-179.024,6.237,148.839
C08511=1173.002,97.065,-51.772,-179.022,6.239,148.839
C08512=1172.997,97.314,-51.790,-179.018,6.240,148.838
C08513=1172.993,97.564,-51.808,-179.016,6.241,148.838
C08514=1172.988,97.813,-51.826,-179.014,6.243,148.837
C08515=1172.983,98.062,-51.844,-179.011,6.243,148.837
C08516=1172.978,98.311,-51.862,-179.008,6.245,148.836
C08517=1172.972,98.561,-51.881,-179.005,6.246,148.836
C08518=1172.968,98.811,-51.899,-179.003,6.247,148.835
C08519=1172.963,99.059,-51.918,-179.000,6.249,148.835
C08520=1172.958,99.308,-51.936,-178.998,6.249,148.834
C08521=1172.953,99.558,-51.954,-178.995,6.251,148.834
C08522=1172.949,99.807,-51.972,-178.992,6.253,148.833
C08523=1172.943,100.057,-51.991,-178.990,6.253,148.833
C08524=1172.939,100.306,-52.009,-178.987,6.255,148.832
C08525=1172.934,100.555,-52.027,-178.984,6.257,148.832
C08526=1172.930,100.804,-52.046,-178.981,6.257,148.831
C08527=1172.925,101.054,-52.064,-178.979,6.259,148.831
C08528=1172.919,101.303,-52.082,-178.977,6.260,148.830
C08529=1172.914,101.552,-52.101,-178.973,6.261,148.830
C08530=1172.910,101.802,-52.119,-178.971,6.263,148.829
C08531=1172.905,102.051,-52.137,-178.969,6.264,148.829
C08532=1172.900,102.300,-52.157,-178.965,6.265,148.828
C08533=1172.895,102.549,-52.175,-178.963,6.267,148.828
C08534=1172.891,102.799,-52.193,-178.961,6.268,148.827
C08535=1172.885,103.048,-52.212,-178.957,6.269,148.827
C08536=1172.880,103.297,-52.230,-178.955,6.271,148.826
C08537=1172.876,103.547,-52.249,-178.952,6.272,148.826
C08538=1172.871,103.796,-52.267,-178.949,6.273,148.825
C08539=1172.866,104.045,-52.286,-178.947,6.274,148.825
C08540=1172.861,104.294,-52.304,-178.944,6.276,148.824
C08541=1172.857,104.543,-52.323,-178.941,6.277,148.824
C08542=1172.851,104.793,-52.342,-178.939,6.278,148.823
C08543=1172.846,105.042,-52.360,-178.936,6.280,148.823
C08544=1172.842,105.291,-52.379,-178.933,6.281,148.822
C08545=1172.837,105.540,-52.397,-178.931,6.282,148.822
C08546=1172.832,105.789,-52.416,-178.928,6.284,148.822
C08547=1172.827,106.058,-52.436,-178.925,6.285,148.821
C08548=1172.822,106.327,-52.456,-178.922,6.287,148.821
C08549=1172.816,106.594,-52.476,-178.919,6.288,148.820
C08550=1172.812,106.863,-52.496,-178.917,6.290,148.819
C08551=1172.806,107.112,-52.515,-178.914,6.291,148.819
C08552=1172.802,107.361,-52.533,-178.911,6.292,148.818
C08553=1172.797,107.611,-52.553,-178.908,6.294,148.818
C08554=1172.792,107.860,-52.571,-178.906,6.295,148.818
C08555=1172.787,108.109,-52.590,-178.903,6.296,148.817
C08556=1172.782,108.359,-52.609,-178.900,6.298,148.817
C08557=1172.778,108.608,-52.627,-178.898,6.299,148.816
C08558=1172.773,108.858,-52.646,-178.895,6.300,148.816
C08559=1172.768,109.106,-52.665,-178.892,6.302,148.815
C08560=1172.762,109.356,-52.684,-178.890,6.303,148.815
C08561=1172.758,109.605,-52.703,-178.887,6.304,148.814
C08562=1172.753,109.854,-52.722,-178.884,6.306,148.814
C08563=1172.749,110.104,-52.740,-178.882,6.307,148.813
C08564=1172.743,110.353,-52.760,-178.880,6.309,148.813
C08565=1172.738,110.602,-52.778,-178.876,6.310,148.812
C08566=1172.734,110.851,-52.797,-178.874,6.311,148.812
C08567=1172.729,111.100,-52.816,-178.871,6.313,148.811
C08568=1172.724,111.350,-52.835,-178.868,6.314,148.811
C08569=1172.719,111.599,-52.854,-178.866,6.316,148.810
C08570=1172.715,111.848,-52.873,-178.863,6.317,148.810
C08571=1172.710,112.097,-52.891,-178.861,6.318,148.810
C08572=1172.705,112.347,-52.911,-178.858,6.320,148.809
C08573=1172.700,112.596,-52.930,-178.855,6.321,148.809
C08574=1172.695,112.845,-52.948,-178.853,6.322,148.808
C08575=1172.691,113.094,-52.967,-178.849,6.324,148.807
C08576=1172.685,113.343,-52.986,-178.847,6.325,148.807
C08577=1172.681,113.593,-53.006,-178.845,6.326,148.807
C08578=1172.676,113.842,-53.024,-178.842,6.328,148.806
C08579=1172.671,114.091,-53.044,-178.839,6.330,148.806
C08580=1172.666,114.340,-53.062,-178.837,6.330,148.805
C08581=1172.662,114.590,-53.082,-178.834,6.332,148.805
C08582=1172.656,114.838,-53.101,-178.831,6.334,148.804
C08583=1172.652,115.088,-53.120,-178.828,6.335,148.804
C08584=1172.647,115.337,-53.139,-178.826,6.336,148.803
C08585=1172.642,115.587,-53.159,-178.823,6.338,148.803
C08586=1172.637,115.835,-53.177,-178.820,6.339,148.802
C08587=1172.633,116.085,-53.197,-178.818,6.340,148.802
C08588=1172.628,116.333,-53.216,-178.815,6.342,148.802
C08589=1172.623,116.584,-53.235,-178.812,6.344,148.801
C08590=1172.618,116.833,-53.254,-178.809,6.345,148.801
C08591=1172.613,117.082,-53.274,-178.807,6.346,148.800
C08592=1172.609,117.331,-53.293,-178.804,6.348,148.800
C08593=1172.603,117.580,-53.312,-178.802,6.349,148.799
C08594=1172.599,117.830,-53.332,-178.798,6.351,148.799
C08595=1172.594,118.078,-53.350,-178.796,6.352,148.798
C08596=1172.589,118.328,-53.370,-178.794,6.353,148.798
C08597=1172.584,118.577,-53.389,-178.791,6.355,148.797
C08598=1172.580,118.826,-53.408,-178.788,6.356,148.797
C08599=1172.575,119.076,-53.428,-178.786,6.357,148.796
C08600=1172.570,119.324,-53.447,-178.783,6.359,148.796
C08601=1172.565,119.574,-53.467,-178.780,6.361,148.796
C08602=1172.561,119.823,-53.486,-178.777,6.363,148.795
C08603=1172.556,120.072,-53.505,-178.775,6.363,148.795
C08604=1172.551,120.321,-53.525,-178.772,6.365,148.794
C08605=1172.546,120.571,-53.544,-178.769,6.367,148.794
C08606=1172.541,120.820,-53.564,-178.767,6.368,148.793
C08607=1172.536,121.069,-53.583,-178.764,6.369,148.793
C08608=1172.532,121.318,-53.602,-178.761,6.371,148.792
C08609=1172.527,121.568,-53.622,-178.759,6.372,148.792
C08610=1172.522,121.817,-53.641,-178.756,6.374,148.792
C08611=1172.517,122.066,-53.661,-178.753,6.375,148.791
C08612=1172.512,122.315,-53.680,-178.751,6.376,148.791
C08613=1172.508,122.564,-53.700,-178.748,6.378,148.790
C08614=1172.503,122.813,-53.720,-178.745,6.380,148.790
C08615=1172.498,123.062,-53.739,-178.743,6.382,148.789
C08616=1172.493,123.312,-53.758,-178.740,6.382,148.789
C08617=1172.488,123.561,-53.778,-178.737,6.384,148.788
C08618=1172.483,123.810,-53.797,-178.735,6.386,148.788
C08619=1172.479,124.059,-53.817,-178.732,6.387,148.788
C08620=1172.474,124.308,-53.837,-178.729,6.389,148.787
C08621=1172.469,124.557,-53.856,-178.727,6.390,148.786
C08622=1172.464,124.807,-53.876,-178.724,6.391,148.786
C08623=1172.460,125.056,-53.895,-178.721,6.393,148.786
C08624=1172.455,125.305,-53.916,-178.718,6.395,148.785
C08625=1172.450,125.554,-53.935,-178.716,6.395,148.785
C08626=1172.445,125.804,-53.955,-178.713,6.397,148.784
C08627=1172.440,126.053,-53.974,-178.710,6.399,148.784
C08628=1172.435,126.302,-53.994,-178.708,6.401,148.783
C08629=1172.431,126.551,-54.014,-178.705,6.402,148.783
C08630=1172.426,126.801,-54.034,-178.702,6.403,148.782
C08631=1172.422,127.049,-54.054,-178.700,6.405,148.782
C08632=1172.417,127.298,-54.073,-178.697,6.406,148.782
C08633=1172.412,127.548,-54.092,-178.694,6.408,148.781
C08634=1172.408,127.797,-54.113,-178.692,6.410,148.781
C08635=1172.403,128.046,-54.133,-178.688,6.411,148.780
C08636=1172.398,128.295,-54.152,-178.686,6.412,148.780
C08637=1172.393,128.544,-54.172,-178.684,6.414,148.779
C08638=1172.388,128.794,-54.192,-178.681,6.416,148.779
C08639=1172.384,129.043,-54.212,-178.678,6.417,148.779
C08640=1172.379,129.292,-54.231,-178.675,6.419,148.778
C08641=1172.374,129.541,-54.251,-178.673,6.420,148.778
C08642=1172.369,129.790,-54.272,-178.670,6.421,148.777
C08643=1172.364,130.040,-54.292,-178.667,6.423,148.777
C08644=1172.359,130.288,-54.312,-178.665,6.425,148.776
C08645=1172.354,130.538,-54.331,-178.662,6.427,148.776
C08646=1172.350,130.787,-54.352,-178.659,6.428,148.775
C08647=1172.345,131.036,-54.371,-178.657,6.429,148.775
C08648=1172.341,131.285,-54.392,-178.654,6.431,148.775
C08649=1172.335,131.534,-54.411,-178.651,6.432,148.774
C08650=1172.331,131.783,-54.432,-178.649,6.434,148.774
C08651=1172.325,132.052,-54.453,-178.645,6.435,148.773
C08652=1172.320,132.321,-54.474,-178.643,6.437,148.773
C08653=1172.315,132.589,-54.497,-178.640,6.439,148.772
C08654=1172.310,132.858,-54.518,-178.637,6.440,148.772
C08655=1172.305,133.107,-54.538,-178.634,6.442,148.771
C08656=1172.301,133.356,-54.558,-178.631,6.444,148.771
C08657=1172.296,133.605,-54.579,-178.629,6.446,148.771
C08658=1172.291,133.855,-54.598,-178.626,6.447,148.770
C08659=1172.286,134.104,-54.619,-178.624,6.448,148.770
C08660=1172.281,134.352,-54.639,-178.621,6.450,148.769
C08661=1172.277,134.602,-54.658,-178.618,6.451,148.769
C08662=1172.272,134.851,-54.679,-178.615,6.453,148.768
C08663=1172.267,135.100,-54.700,-178.613,6.455,148.768
C08664=1172.262,135.350,-54.719,-178.610,6.457,148.768
C08665=1172.258,135.598,-54.740,-178.607,6.458,148.767
C08666=1172.253,135.847,-54.760,-178.605,6.459,148.767
C08667=1172.248,136.097,-54.780,-178.602,6.461,148.767
C08668=1172.243,136.346,-54.800,-178.599,6.462,148.766
C08669=1172.238,136.595,-54.821,-178.597,6.464,148.766
C08670=1172.234,136.844,-54.840,-178.594,6.466,148.765
C08671=1172.228,137.093,-54.861,-178.591,6.468,148.765
C08672=1172.224,137.342,-54.882,-178.588,6.469,148.764
C08673=1172.220,137.591,-54.902,-178.586,6.471,148.764
C08674=1172.215,137.841,-54.922,-178.584,6.472,148.764
C08675=1172.210,138.090,-54.943,-178.580,6.473,148.763
C08676=1172.205,138.339,-54.963,-178.578,6.475,148.763
C08677=1172.201,138.588,-54.984,-178.575,6.477,148.762
C08678=1172.196,138.837,-55.005,-178.572,6.479,148.762
C08679=1172.191,139.086,-55.025,-178.570,6.480,148.761
C08680=1172.186,139.336,-55.045,-178.567,6.482,148.761
C08681=1172.182,139.585,-55.065,-178.564,6.484,148.761
C08682=1172.177,139.834,-55.086,-178.562,6.486,148.760
C08683=1172.172,140.083,-55.106,-178.559,6.486,148.760
C08684=1172.167,140.332,-55.127,-178.556,6.488,148.759
C08685=1172.162,140.580,-55.147,-178.554,6.490,148.759
C08686=1172.158,140.829,-55.168,-178.551,6.491,148.758
C08687=1172.153,141.079,-55.189,-178.548,6.493,148.758
C08688=1172.148,141.328,-55.208,-178.545,6.495,148.758
C08689=1172.143,141.577,-55.229,-178.543,6.497,148.757
C08690=1172.138,141.826,-55.250,-178.540,6.498,148.757
C08691=1172.134,142.075,-55.270,-178.537,6.500,148.757
C08692=1172.129,142.325,-55.291,-178.535,6.502,148.756
C08693=1172.125,142.574,-55.312,-178.531,6.503,148.756
C08694=1172.120,142.823,-55.332,-178.529,6.504,148.755
C08695=1172.115,143.072,-55.353,-178.527,6.506,148.755
C08696=1172.111,143.321,-55.373,-178.524,6.508,148.754
C08697=1172.106,143.571,-55.394,-178.521,6.509,148.754
C08698=1172.101,143.820,-55.415,-178.519,6.511,148.754
C08699=1172.096,144.069,-55.436,-178.516,6.513,148.753
C08700=1172.092,144.318,-55.456,-178.513,6.515,148.753
C08701=1172.087,144.566,-55.478,-178.510,6.516,148.752
C08702=1172.082,144.815,-55.498,-178.508,6.518,148.752
C08703=1172.078,145.064,-55.518,-178.505,6.520,148.752
C08704=1172.073,145.314,-55.539,-178.502,6.522,148.751
C08705=1172.068,145.563,-55.560,-178.499,6.523,148.751
C08706=1172.063,145.812,-55.581,-178.496,6.525,148.750
C08707=1172.058,146.061,-55.602,-178.494,6.526,148.750
C08708=1172.053,146.310,-55.622,-178.492,6.527,148.750
C08709=1172.049,146.560,-55.643,-178.489,6.529,148.749
C08710=1172.045,146.808,-55.665,-178.486,6.531,148.749
C08711=1172.039,147.058,-55.685,-178.484,6.533,148.748
C08712=1172.035,147.307,-55.706,-178.481,6.534,148.748
C08713=1172.030,147.556,-55.727,-178.478,6.536,148.748
C08714=1172.025,147.805,-55.747,-178.475,6.538,148.747
C08715=1172.021,148.053,-55.769,-178.473,6.540,148.747
C08716=1172.015,148.303,-55.790,-178.470,6.541,148.746
C08717=1172.011,148.552,-55.810,-178.467,6.543,148.746
C08718=1172.006,148.802,-55.832,-178.465,6.545,148.746
C08719=1172.002,149.050,-55.853,-178.462,6.547,148.745
C08720=1171.997,149.299,-55.874,-178.459,6.548,148.745
C08721=1171.992,149.548,-55.895,-178.456,6.550,148.744
C08722=1171.987,149.797,-55.915,-178.453,6.552,148.744
C08723=1171.983,150.046,-55.937,-178.451,6.553,148.744
C08724=1171.977,150.295,-55.958,-178.448,6.555,148.743
C08725=1171.974,150.545,-55.978,-178.445,6.557,148.743
C08726=1171.969,150.794,-56.000,-178.443,6.559,148.742
C08727=1171.964,151.043,-56.021,-178.440,6.560,148.742
C08728=1171.959,151.292,-56.041,-178.437,6.562,148.742
C08729=1171.954,151.540,-56.063,-178.435,6.564,148.741
C08730=1171.950,151.790,-56.084,-178.432,6.566,148.741
C08731=1171.946,152.039,-56.105,-178.429,6.567,148.741
C08732=1171.940,152.288,-56.126,-178.427,6.569,148.740
C08733=1171.935,152.537,-56.147,-178.424,6.571,148.740
C08734=1171.930,152.786,-56.169,-178.421,6.573,148.739
C08735=1171.926,153.035,-56.190,-178.418,6.574,148.739
C08736=1171.922,153.284,-56.211,-178.416,6.576,148.739
C08737=1171.916,153.533,-56.232,-178.413,6.578,148.738
C08738=1171.912,153.782,-56.254,-178.410,6.580,148.738
C08739=1171.907,154.031,-56.274,-178.408,6.581,148.738
C08740=1171.903,154.280,-56.297,-178.405,6.583,148.737
C08741=1171.898,154.530,-56.318,-178.402,6.585,148.737
C08742=1171.893,154.778,-56.339,-178.400,6.587,148.736
C08743=1171.888,155.027,-56.360,-178.397,6.588,148.736
C08744=1171.884,155.277,-56.382,-178.394,6.590,148.736
C08745=1171.879,155.526,-56.403,-178.392,6.592,148.735
C08746=1171.874,155.774,-56.424,-178.389,6.594,148.735
C08747=1171.869,156.024,-56.445,-178.386,6.595,148.735
C08748=1171.865,156.273,-56.467,-178.383,6.597,148.734
C08749=1171.860,156.521,-56.488,-178.381,6.599,148.734
C08750=1171.855,156.771,-56.509,-178.378,6.601,148.733
C08751=1171.851,157.020,-56.531,-178.375,6.602,148.733
C08752=1171.846,157.269,-56.552,-178.373,6.604,148.733
C08753=1171.841,157.518,-56.574,-178.370,6.606,148.732
C08754=1171.836,157.766,-56.596,-178.367,6.608,148.732
C08755=1171.831,158.036,-56.618,-178.365,6.609,148.732
C08756=1171.826,158.305,-56.642,-178.361,6.611,148.731
C08757=1171.821,158.573,-56.665,-178.359,6.613,148.731
C08758=1171.816,158.843,-56.689,-178.355,6.615,148.730
C08759=1171.812,159.092,-56.711,-178.353,6.617,148.730
C08760=1171.807,159.341,-56.731,-178.350,6.619,148.729
C08761=1171.802,159.590,-56.753,-178.347,6.620,148.729
C08762=1171.798,159.839,-56.775,-178.345,6.622,148.729
C08763=1171.793,160.088,-56.796,-178.342,6.624,148.728
C08764=1171.788,160.337,-56.817,-178.339,6.626,148.728
C08765=1171.784,160.586,-56.840,-178.337,6.627,148.728
C08766=1171.779,160.835,-56.861,-178.334,6.629,148.727
C08767=1171.774,161.083,-56.883,-178.331,6.631,148.727
C08768=1171.770,161.333,-56.904,-178.329,6.633,148.726
C08769=1171.765,161.582,-56.926,-178.326,6.634,148.726
C08770=1171.760,161.831,-56.948,-178.323,6.636,148.726
C08771=1171.756,162.080,-56.970,-178.321,6.638,148.725
C08772=1171.751,162.329,-56.991,-178.318,6.640,148.725
C08773=1171.746,162.578,-57.013,-178.316,6.642,148.725
C08774=1171.741,162.827,-57.034,-178.313,6.644,148.724
C08775=1171.737,163.077,-57.056,-178.310,6.646,148.724
C08776=1171.732,163.325,-57.078,-178.307,6.648,148.724
C08777=1171.727,163.574,-57.100,-178.304,6.650,148.723
C08778=1171.723,163.823,-57.122,-178.302,6.651,148.723
C08779=1171.718,164.072,-57.143,-178.299,6.653,148.723
C08780=1171.714,164.321,-57.166,-178.296,6.655,148.722
C08781=1171.709,164.570,-57.187,-178.294,6.657,148.722
C08782=1171.704,164.820,-57.210,-178.291,6.658,148.721
C08783=1171.699,165.068,-57.232,-178.288,6.660,148.721
C08784=1171.694,165.317,-57.253,-178.285,6.662,148.721
C08785=1171.690,165.566,-57.275,-178.283,6.664,148.720
C08786=1171.685,165.815,-57.297,-178.280,6.665,148.720
C08787=1171.681,166.064,-57.319,-178.277,6.667,148.720
C08788=1171.676,166.313,-57.341,-178.275,6.669,148.719
C08789=1171.672,166.562,-57.363,-178.271,6.672,148.719
C08790=1171.667,166.811,-57.384,-178.269,6.673,148.719
C08791=1171.662,167.060,-57.407,-178.267,6.675,148.718
C08792=1171.657,167.309,-57.429,-178.264,6.677,148.718
C08793=1171.653,167.558,-57.451,-178.261,6.679,148.718
C08794=1171.648,167.807,-57.472,-178.259,6.681,148.717
C08795=1171.644,168.056,-57.495,-178.256,6.682,148.717
C08796=1171.639,168.304,-57.517,-178.253,6.684,148.717
C08797=1171.634,168.554,-57.540,-178.250,6.686,148.716
C08798=1171.629,168.803,-57.561,-178.248,6.688,148.716
C08799=1171.625,169.052,-57.583,-178.245,6.690,148.715
C08800=1171.620,169.301,-57.605,-178.242,6.692,148.715
C08801=1171.615,169.550,-57.628,-178.239,6.694,148.715
C08802=1171.610,169.798,-57.650,-178.236,6.696,148.714
C08803=1171.606,170.048,-57.672,-178.234,6.698,148.714
C08804=1171.601,170.296,-57.694,-178.232,6.699,148.714
C08805=1171.596,170.546,-57.716,-178.229,6.701,148.713
C08806=1171.592,170.795,-57.738,-178.226,6.703,148.713
C08807=1171.587,171.043,-57.761,-178.224,6.705,148.713
C08808=1171.583,171.293,-57.783,-178.221,6.707,148.712
C08809=1171.577,171.542,-57.805,-178.218,6.709,148.712
C08810=1171.574,171.790,-57.828,-178.215,6.711,148.712
C08811=1171.569,172.039,-57.850,-178.212,6.713,148.711
C08812=1171.564,172.289,-57.872,-178.210,6.714,148.711
C08813=1171.559,172.538,-57.894,-178.207,6.717,148.711
C08814=1171.555,172.786,-57.917,-178.205,6.718,148.710
C08815=1171.550,173.036,-57.939,-178.202,6.720,148.710
C08816=1171.545,173.284,-57.961,-178.199,6.722,148.710
C08817=1171.541,173.533,-57.984,-178.196,6.724,148.709
C08818=1171.536,173.783,-58.006,-178.193,6.726,148.709
C08819=1171.531,174.031,-58.029,-178.191,6.728,148.709
C08820=1171.526,174.280,-58.051,-178.188,6.730,148.708
C08821=1171.522,174.529,-58.073,-178.186,6.732,148.708
C08822=1171.518,174.778,-58.096,-178.183,6.734,148.708
C08823=1171.513,175.027,-58.119,-178.180,6.735,148.707
C08824=1171.508,175.275,-58.141,-178.177,6.738,148.707
C08825=1171.503,175.525,-58.164,-178.174,6.740,148.707
C08826=1171.499,175.774,-58.186,-178.172,6.741,148.706
C08827=1171.494,176.022,-58.208,-178.169,6.743,148.706
C08828=1171.489,176.271,-58.231,-178.167,6.745,148.706
C08829=1171.485,176.521,-58.253,-178.164,6.747,148.705
C08830=1171.480,176.769,-58.276,-178.161,6.750,148.705
C08831=1171.476,177.018,-58.298,-178.158,6.751,148.705
C08832=1171.471,177.267,-58.322,-178.156,6.753,148.704
C08833=1171.466,177.516,-58.344,-178.153,6.755,148.704
C08834=1171.461,177.765,-58.367,-178.150,6.757,148.704
C08835=1171.457,178.014,-58.389,-178.148,6.759,148.704
C08836=1171.452,178.264,-58.412,-178.145,6.761,148.703
C08837=1171.448,178.512,-58.434,-178.142,6.763,148.703
C08838=1171.443,178.761,-58.457,-178.139,6.765,148.702
C08839=1171.439,179.010,-58.480,-178.137,6.767,148.702
C08840=1171.433,179.259,-58.502,-178.134,6.768,148.702
C08841=1171.429,179.508,-58.525,-178.132,6.771,148.702
C08842=1171.425,179.757,-58.549,-178.129,6.773,148.701
C08843=1171.420,180.006,-58.571,-178.126,6.775,148.701
C08844=1171.415,180.254,-58.594,-178.123,6.777,148.701
C08845=1171.411,180.503,-58.616,-178.121,6.778,148.700
C08846=1171.406,180.753,-58.639,-178.118,6.780,148.700
C08847=1171.402,181.001,-58.662,-178.116,6.782,148.700
C08848=1171.397,181.250,-58.685,-178.112,6.785,148.699
C08849=1171.392,181.499,-58.707,-178.110,6.787,148.699
C08850=1171.388,181.748,-58.730,-178.107,6.789,148.699
C08851=1171.383,181.997,-58.753,-178.104,6.790,148.698
C08852=1171.378,182.246,-58.777,-178.102,6.792,148.698
C08853=1171.374,182.494,-58.799,-178.099,6.795,148.698
C08854=1171.369,182.744,-58.822,-178.096,6.797,148.697
C08855=1171.365,182.993,-58.845,-178.094,6.799,148.697
C08856=1171.360,183.242,-58.868,-178.091,6.800,148.697
C08857=1171.356,183.491,-58.891,-178.088,6.802,148.696
C08858=1171.351,183.739,-58.914,-178.085,6.805,148.696
C08859=1171.346,184.008,-58.939,-178.083,6.807,148.696
C08860=1171.340,184.278,-58.964,-178.079,6.809,148.696
C08861=1171.336,184.548,-58.988,-178.077,6.811,148.695
C08862=1171.330,184.817,-59.013,-178.074,6.814,148.695
C08863=1171.326,185.066,-59.037,-178.071,6.815,148.694
C08864=1171.322,185.315,-59.059,-178.068,6.817,148.694
C08865=1171.317,185.564,-59.083,-178.065,6.819,148.694
C08866=1171.312,185.813,-59.106,-178.063,6.821,148.694
C08867=1171.308,186.062,-59.129,-178.060,6.824,148.693
C08868=1171.304,186.311,-59.152,-178.057,6.826,148.693
C08869=1171.298,186.559,-59.175,-178.055,6.827,148.693
C08870=1171.294,186.808,-59.199,-178.052,6.829,148.692
C08871=1171.289,187.057,-59.222,-178.049,6.832,148.692
C08872=1171.285,187.306,-59.245,-178.047,6.834,148.692
C08873=1171.280,187.555,-59.268,-178.044,6.836,148.691
C08874=1171.276,187.804,-59.291,-178.041,6.837,148.691
C08875=1171.271,188.053,-59.315,-178.038,6.840,148.691
C08876=1171.266,188.302,-59.338,-178.036,6.842,148.691
C08877=1171.262,188.551,-59.361,-178.033,6.844,148.690
C08878=1171.257,188.799,-59.384,-178.030,6.846,148.690
C08879=1171.252,189.048,-59.407,-178.028,6.848,148.690
C08880=1171.248,189.297,-59.431,-178.025,6.850,148.689
C08881=1171.243,189.546,-59.454,-178.022,6.852,148.689
C08882=1171.238,189.795,-59.477,-178.020,6.854,148.689
C08883=1171.233,190.044,-59.501,-178.017,6.856,148.689
C08884=1171.229,190.293,-59.523,-178.014,6.859,148.688
C08885=1171.225,190.542,-59.548,-178.011,6.860,148.688
C08886=1171.220,190.791,-59.571,-178.009,6.862,148.688
C08887=1171.216,191.040,-59.594,-178.006,6.865,148.687
C08888=1171.211,191.289,-59.618,-178.003,6.867,148.687
C08889=1171.206,191.538,-59.641,-178.001,6.869,148.687
C08890=1171.202,191.786,-59.665,-177.998,6.870,148.686
C08891=1171.197,192.035,-59.688,-177.995,6.873,148.686
C08892=1171.193,192.284,-59.712,-177.993,6.875,148.686
C08893=1171.188,192.533,-59.735,-177.990,6.877,148.686
C08894=1171.183,192.782,-59.759,-177.987,6.879,148.685
C08895=1171.179,193.031,-59.783,-177.984,6.882,148.685
C08896=1171.174,193.280,-59.806,-177.982,6.883,148.685
C08897=1171.169,193.529,-59.829,-177.979,6.885,148.684
C08898=1171.165,193.777,-59.853,-177.977,6.887,148.684
C08899=1171.160,194.026,-59.877,-177.974,6.890,148.684
C08900=1171.156,194.275,-59.900,-177.971,6.892,148.684
C08901=1171.151,194.524,-59.924,-177.968,6.893,148.683
C08902=1171.146,194.773,-59.948,-177.965,6.896,148.683
C08903=1171.142,195.022,-59.971,-177.963,6.898,148.683
C08904=1171.137,195.270,-59.995,-177.960,6.900,148.682
C08905=1171.133,195.519,-60.018,-177.958,6.902,148.682
C08906=1171.128,195.768,-60.042,-177.955,6.905,148.682
C08907=1171.124,196.017,-60.066,-177.952,6.906,148.682
C08908=1171.119,196.266,-60.089,-177.949,6.908,148.681
C08909=1171.114,196.514,-60.113,-177.947,6.911,148.681
C08910=1171.110,196.763,-60.137,-177.944,6.913,148.681
C08911=1171.105,197.011,-60.161,-177.941,6.915,148.680
C08912=1171.101,197.260,-60.184,-177.938,6.918,148.680
C08913=1171.096,197.509,-60.208,-177.936,6.919,148.680
C08914=1171.092,197.758,-60.231,-177.933,6.921,148.680
C08915=1171.086,198.007,-60.256,-177.930,6.924,148.680
C08916=1171.082,198.256,-60.280,-177.928,6.926,148.679
C08917=1171.078,198.505,-60.304,-177.925,6.928,148.679
C08918=1171.073,198.754,-60.327,-177.922,6.929,148.679
C08919=1171.069,199.002,-60.351,-177.920,6.932,148.678
C08920=1171.064,199.251,-60.375,-177.917,6.934,148.678
C08921=1171.060,199.500,-60.399,-177.914,6.936,148.678
C08922=1171.054,199.749,-60.423,-177.911,6.939,148.678
C08923=1171.050,199.997,-60.447,-177.909,6.941,148.677
C08924=1171.046,200.247,-60.471,-177.906,6.942,148.677
C08925=1171.041,200.496,-60.495,-177.903,6.945,148.677
C08926=1171.037,200.744,-60.519,-177.901,6.947,148.676
C08927=1171.032,200.993,-60.543,-177.898,6.949,148.676
C08928=1171.027,201.242,-60.567,-177.895,6.952,148.676
C08929=1171.023,201.490,-60.591,-177.893,6.954,148.676
C08930=1171.019,201.739,-60.615,-177.890,6.955,148.675
C08931=1171.014,201.988,-60.639,-177.887,6.958,148.675
C08932=1171.009,202.237,-60.663,-177.884,6.960,148.675
C08933=1171.005,202.485,-60.687,-177.882,6.962,148.675
C08934=1171.000,202.734,-60.711,-177.879,6.965,148.674
C08935=1170.996,202.983,-60.735,-177.876,6.967,148.674
C08936=1170.991,203.232,-60.760,-177.874,6.968,148.674
C08937=1170.987,203.481,-60.784,-177.871,6.971,148.674
C08938=1170.982,203.729,-60.808,-177.868,6.973,148.673
C08939=1170.977,203.978,-60.832,-177.866,6.975,148.673
C08940=1170.973,204.227,-60.856,-177.863,6.978,148.673
C08941=1170.969,204.476,-60.880,-177.860,6.980,148.673
C08942=1170.964,204.725,-60.905,-177.857,6.983,148.672
C08943=1170.959,204.973,-60.929,-177.855,6.984,148.672
C08944=1170.955,205.222,-60.952,-177.852,6.986,148.672
C08945=1170.950,205.472,-60.978,-177.849,6.989,148.672
C08946=1170.946,205.720,-61.002,-177.847,6.991,148.671
C08947=1170.941,205.968,-61.026,-177.844,6.993,148.671
C08948=1170.936,206.217,-61.050,-177.841,6.996,148.671
C08949=1170.932,206.466,-61.075,-177.838,6.997,148.670
C08950=1170.927,206.715,-61.099,-177.836,6.999,148.670
C08951=1170.923,206.963,-61.124,-177.833,7.002,148.670
C08952=1170.918,207.212,-61.148,-177.830,7.004,148.670
C08953=1170.914,207.461,-61.173,-177.828,7.007,148.670
C08954=1170.909,207.710,-61.197,-177.825,7.009,148.669
C08955=1170.904,207.958,-61.221,-177.823,7.011,148.669
C08956=1170.901,208.207,-61.246,-177.819,7.013,148.669
C08957=1170.895,208.456,-61.270,-177.817,7.015,148.668
C08958=1170.891,208.705,-61.295,-177.815,7.017,148.668
C08959=1170.886,208.953,-61.319,-177.811,7.020,148.668
C08960=1170.882,209.202,-61.344,-177.809,7.022,148.668
C08961=1170.877,209.451,-61.368,-177.806,7.025,148.668
C08962=1170.873,209.700,-61.392,-177.803,7.026,148.667
C08963=1170.868,209.970,-61.419,-177.800,7.029,148.667
C08964=1170.863,210.241,-61.446,-177.798,7.031,148.667
C08965=1170.857,210.511,-61.472,-177.795,7.034,148.667
C08966=1170.853,210.782,-61.499,-177.791,7.036,148.666
C08967=1170.848,211.031,-61.523,-177.789,7.038,148.666
C08968=1170.844,211.279,-61.549,-177.786,7.041,148.666
C08969=1170.840,211.528,-61.573,-177.784,7.043,148.666
C08970=1170.835,211.777,-61.598,-177.781,7.045,148.665
C08971=1170.830,212.026,-61.623,-177.778,7.048,148.665
C08972=1170.826,212.274,-61.647,-177.776,7.050,148.665
C08973=1170.821,212.523,-61.672,-177.772,7.052,148.665
C08974=1170.817,212.772,-61.697,-177.770,7.054,148.664
C08975=1170.812,213.020,-61.721,-177.767,7.057,148.664
C08976=1170.807,213.270,-61.746,-177.765,7.059,148.664
C08977=1170.803,213.518,-61.771,-177.762,7.061,148.664
C08978=1170.798,213.766,-61.796,-177.759,7.064,148.664
C08979=1170.794,214.015,-61.820,-177.757,7.066,148.663
C08980=1170.789,214.264,-61.845,-177.753,7.068,148.663
C08981=1170.785,214.513,-61.871,-177.751,7.070,148.663
C08982=1170.781,214.761,-61.895,-177.749,7.072,148.662
C08983=1170.776,215.011,-61.920,-177.746,7.075,148.662
C08984=1170.771,215.260,-61.945,-177.743,7.077,148.662
C08985=1170.767,215.507,-61.969,-177.740,7.080,148.662
C08986=1170.762,215.757,-61.994,-177.738,7.082,148.662
C08987=1170.758,216.005,-62.020,-177.735,7.085,148.662
C08988=1170.754,216.254,-62.044,-177.732,7.086,148.661
C08989=1170.749,216.503,-62.069,-177.730,7.089,148.661
C08990=1170.744,216.752,-62.095,-177.727,7.091,148.661
C08991=1170.739,217.000,-62.119,-177.724,7.093,148.660
C08992=1170.736,217.249,-62.144,-177.721,7.096,148.660
C08993=1170.731,217.497,-62.169,-177.719,7.098,148.660
C08994=1170.726,217.746,-62.195,-177.716,7.101,148.660
C08995=1170.721,217.995,-62.220,-177.713,7.102,148.660
C08996=1170.718,218.244,-62.244,-177.711,7.105,148.660
C08997=1170.713,218.492,-62.269,-177.708,7.107,148.659
C08998=1170.708,218.741,-62.295,-177.705,7.110,148.659
C08999=1170.703,218.990,-62.320,-177.702,7.112,148.659
C09000=1170.700,219.238,-62.345,-177.700,7.115,148.659
C09001=1170.695,219.487,-62.370,-177.697,7.117,148.658
C09002=1170.691,219.736,-62.395,-177.695,7.119,148.658
C09003=1170.685,219.984,-62.420,-177.692,7.121,148.658
C09004=1170.681,220.233,-62.446,-177.689,7.123,148.658
C09005=1170.676,220.482,-62.470,-177.686,7.126,148.657
C09006=1170.673,220.730,-62.496,-177.684,7.128,148.657
C09007=1170.668,220.979,-62.521,-177.681,7.131,148.657
C09008=1170.663,221.228,-62.546,-177.679,7.133,148.657
C09009=1170.659,221.477,-62.572,-177.675,7.136,148.657
C09010=1170.654,221.725,-62.597,-177.673,7.138,148.657
C09011=1170.650,221.974,-62.622,-177.670,7.140,148.656
C09012=1170.645,222.222,-62.648,-177.668,7.142,148.656
C09013=1170.641,222.471,-62.673,-177.665,7.145,148.656
C09014=1170.637,222.720,-62.698,-177.662,7.147,148.656
C09015=1170.632,222.968,-62.723,-177.659,7.150,148.655
C09016=1170.628,223.217,-62.749,-177.657,7.152,148.655
C09017=1170.623,223.466,-62.774,-177.654,7.155,148.655
C09018=1170.618,223.715,-62.799,-177.651,7.157,148.655
C09019=1170.614,223.964,-62.825,-177.648,7.159,148.655
C09020=1170.609,224.212,-62.850,-177.646,7.161,148.654
C09021=1170.605,224.461,-62.876,-177.643,7.164,148.654
C09022=1170.600,224.709,-62.901,-177.641,7.166,148.654
C09023=1170.596,224.958,-62.927,-177.638,7.169,148.654
C09024=1170.591,225.207,-62.952,-177.635,7.171,148.654
C09025=1170.587,225.455,-62.978,-177.632,7.174,148.654
C09026=1170.582,225.704,-63.004,-177.630,7.176,148.653
C09027=1170.578,225.953,-63.029,-177.627,7.179,148.653
C09028=1170.573,226.201,-63.054,-177.624,7.180,148.653
C09029=1170.569,226.450,-63.080,-177.622,7.183,148.653
C09030=1170.565,226.699,-63.105,-177.619,7.185,148.652
C09031=1170.560,226.947,-63.131,-177.616,7.188,148.652
C09032=1170.556,227.196,-63.157,-177.614,7.190,148.652
C09033=1170.551,227.445,-63.182,-177.611,7.193,148.652
C09034=1170.547,227.693,-63.208,-177.609,7.195,148.652
C09035=1170.542,227.942,-63.234,-177.605,7.198,148.651
C09036=1170.537,228.191,-63.260,-177.603,7.200,148.651
C09037=1170.533,228.439,-63.285,-177.600,7.202,148.651
C09038=1170.528,228.688,-63.311,-177.598,7.204,148.651
C09039=1170.524,228.936,-63.337,-177.595,7.207,148.651
C09040=1170.520,229.185,-63.362,-177.592,7.210,148.651
C09041=1170.515,229.433,-63.388,-177.590,7.212,148.650
C09042=1170.511,229.682,-63.414,-177.586,7.215,148.650
C09043=1170.507,229.931,-63.439,-177.584,7.217,148.650
C09044=1170.502,230.180,-63.466,-177.581,7.220,148.650
C09045=1170.497,230.428,-63.491,-177.579,7.222,148.650
C09046=1170.493,230.677,-63.517,-177.576,7.225,148.650
C09047=1170.488,230.926,-63.543,-177.573,7.226,148.649
C09048=1170.484,231.174,-63.569,-177.571,7.229,148.649
C09049=1170.479,231.422,-63.595,-177.568,7.231,148.649
C09050=1170.475,231.671,-63.621,-177.565,7.234,148.649
C09051=1170.470,231.920,-63.647,-177.562,7.237,148.649
C09052=1170.466,232.169,-63.672,-177.560,7.239,148.648
C09053=1170.461,232.417,-63.698,-177.557,7.242,148.648
C09054=1170.457,232.665,-63.725,-177.554,7.244,148.648
C09055=1170.452,232.914,-63.750,-177.552,7.247,148.648
C09056=1170.448,233.163,-63.776,-177.549,7.249,148.648
C09057=1170.444,233.412,-63.802,-177.546,7.251,148.647
C09058=1170.438,233.660,-63.828,-177.543,7.254,148.647
C09059=1170.435,233.908,-63.854,-177.541,7.256,148.647
C09060=1170.430,234.157,-63.880,-177.538,7.259,148.647
C09061=1170.425,234.406,-63.907,-177.536,7.261,148.647
C09062=1170.421,234.654,-63.933,-177.533,7.264,148.647
C09063=1170.417,234.903,-63.959,-177.530,7.266,148.647
C09064=1170.412,235.152,-63.985,-177.528,7.269,148.646
C09065=1170.408,235.400,-64.011,-177.524,7.271,148.646
C09066=1170.404,235.649,-64.037,-177.522,7.274,148.646
C09067=1170.398,235.921,-64.066,-177.519,7.277,148.646
C09068=1170.394,236.192,-64.094,-177.516,7.279,148.646
C09069=1170.389,236.464,-64.122,-177.513,7.282,148.646
C09070=1170.384,236.736,-64.152,-177.510,7.285,148.645
C09071=1170.380,236.984,-64.177,-177.508,7.287,148.645
C09072=1170.374,237.232,-64.204,-177.505,7.290,148.645
C09073=1170.370,237.481,-64.230,-177.502,7.292,148.645
C09074=1170.366,237.729,-64.256,-177.500,7.295,148.645
C09075=1170.361,237.978,-64.283,-177.497,7.298,148.645
C09076=1170.357,238.227,-64.309,-177.494,7.299,148.644
C09077=1170.352,238.476,-64.336,-177.492,7.302,148.644
C09078=1170.348,238.724,-64.362,-177.489,7.305,148.644
C09079=1170.344,238.973,-64.388,-177.486,7.307,148.644
C09080=1170.340,239.221,-64.415,-177.484,7.310,148.644
C09081=1170.335,239.470,-64.441,-177.481,7.313,148.644
C09082=1170.331,239.718,-64.468,-177.478,7.315,148.643
C09083=1170.326,239.967,-64.493,-177.475,7.318,148.643
C09084=1170.321,240.215,-64.520,-177.473,7.320,148.643
C09085=1170.317,240.463,-64.547,-177.470,7.323,148.643
C09086=1170.312,240.712,-64.573,-177.467,7.325,148.643
C09087=1170.308,240.961,-64.599,-177.465,7.328,148.643
C09088=1170.303,241.210,-64.626,-177.462,7.331,148.643
C09089=1170.300,241.458,-64.652,-177.459,7.333,148.642
C09090=1170.295,241.706,-64.679,-177.457,7.335,148.642
C09091=1170.290,241.955,-64.706,-177.454,7.338,148.642
C09092=1170.286,242.204,-64.732,-177.451,7.340,148.642
C09093=1170.281,242.452,-64.759,-177.449,7.343,148.642
C09094=1170.277,242.701,-64.785,-177.446,7.346,148.642
C09095=1170.272,242.949,-64.812,-177.444,7.348,148.642
C09096=1170.269,243.198,-64.838,-177.440,7.351,148.641
C09097=1170.264,243.446,-64.865,-177.438,7.354,148.641
C09098=1170.259,243.695,-64.892,-177.436,7.356,148.641
C09099=1170.255,243.943,-64.918,-177.432,7.358,148.641
C09100=1170.250,244.192,-64.945,-177.430,7.361,148.641
C09101=1170.246,244.440,-64.972,-177.427,7.364,148.641
C09102=1170.242,244.689,-64.999,-177.425,7.367,148.641
C09103=1170.237,244.938,-65.025,-177.422,7.368,148.640
C09104=1170.233,245.186,-65.052,-177.419,7.371,148.640
C09105=1170.229,245.435,-65.079,-177.416,7.374,148.640
C09106=1170.224,245.684,-65.106,-177.414,7.376,148.640
C09107=1170.220,245.932,-65.133,-177.411,7.379,148.640
C09108=1170.216,246.180,-65.160,-177.408,7.382,148.640
C09109=1170.211,246.429,-65.187,-177.406,7.384,148.640
C09110=1170.206,246.678,-65.213,-177.403,7.387,148.640
C09111=1170.202,246.926,-65.240,-177.401,7.390,148.640
C09112=1170.197,247.175,-65.267,-177.398,7.392,148.639
C09113=1170.193,247.423,-65.294,-177.395,7.395,148.639
C09114=1170.189,247.671,-65.320,-177.392,7.398,148.639
C09115=1170.184,247.920,-65.347,-177.390,7.400,148.639
C09116=1170.180,248.168,-65.374,-177.387,7.403,148.639
C09117=1170.175,248.417,-65.402,-177.384,7.405,148.639
C09118=1170.172,248.666,-65.428,-177.382,7.408,148.639
C09119=1170.167,248.914,-65.455,-177.379,7.411,148.638
C09120=1170.162,249.163,-65.482,-177.377,7.414,148.638
C09121=1170.158,249.411,-65.509,-177.373,7.416,148.638
C09122=1170.153,249.660,-65.536,-177.371,7.418,148.638
C09123=1170.149,249.908,-65.563,-177.368,7.421,148.638
C09124=1170.145,250.156,-65.591,-177.366,7.424,148.638
C09125=1170.141,250.405,-65.618,-177.364,7.426,148.638
C09126=1170.136,250.653,-65.645,-177.360,7.429,148.638
C09127=1170.131,250.902,-65.672,-177.358,7.432,148.637
C09128=1170.127,251.150,-65.699,-177.355,7.434,148.637
C09129=1170.122,251.399,-65.726,-177.353,7.437,148.637
C09130=1170.118,251.647,-65.753,-177.350,7.440,148.637
C09131=1170.114,251.896,-65.780,-177.347,7.442,148.637
C09132=1170.110,252.144,-65.808,-177.344,7.445,148.637
C09133=1170.105,252.393,-65.835,-177.342,7.448,148.637
C09134=1170.100,252.641,-65.862,-177.339,7.451,148.637
C09135=1170.096,252.890,-65.889,-177.337,7.453,148.637
C09136=1170.092,253.138,-65.917,-177.334,7.456,148.637
C09137=1170.087,253.387,-65.944,-177.331,7.458,148.636
C09138=1170.083,253.635,-65.971,-177.329,7.461,148.636
C09139=1170.078,253.884,-65.999,-177.326,7.464,148.636
C09140=1170.074,254.132,-66.027,-177.323,7.466,148.636
C09141=1170.070,254.381,-66.054,-177.320,7.469,148.636
C09142=1170.065,254.629,-66.081,-177.318,7.472,148.636
C09143=1170.061,254.877,-66.108,-177.315,7.475,148.636
C09144=1170.057,255.126,-66.135,-177.312,7.477,148.636
